LIN {X 0,Y 337.966,Z 536.674,A -85,B 0,C 180,E1 16019.152,E2 16019.152} C_VEL
LIN {X 0,Y 337.966,Z 536.674,A -85,B 0,C 180,E1 16014.908,E2 16014.908} C_VEL
LIN {X 0,Y 337.973,Z 536.675,A -85,B 0,C 180,E1 16010.807,E2 16010.807} C_VEL
LIN {X 0,Y 337.973,Z 536.677,A -85,B 0,C 180,E1 16006.484,E2 16006.484} C_VEL
LIN {X 0,Y 337.975,Z 536.732,A -85,B 0,C 180,E1 16002.259,E2 16002.259} C_VEL
LIN {X 0,Y 338.082,Z 537.452,A -85,B 0,C 180,E1 16001.73,E2 16001.73} C_VEL
LIN {X 0,Y 340.143,Z 542.274,A -85,B 0,C 180,E1 15999.651,E2 15999.651} C_VEL
LIN {X 0,Y 341.904,Z 546.345,A -85,B 0,C 180,E1 15998.017,E2 15998.017} C_VEL
LIN {X 0,Y 344.615,Z 552.699,A -85,B 0,C 180,E1 15995.632,E2 15995.632} C_VEL
LIN {X 0,Y 348.357,Z 562.803,A -85,B 0,C 180,E1 15992.291,E2 15992.291} C_VEL
LIN {X 0,Y 352.153,Z 574.379,A -85,B 0,C 180,E1 15988.885,E2 15988.885} C_VEL
LIN {X 0,Y 355.607,Z 586.974,A -85,B 0,C 180,E1 15985.587,E2 15985.587} C_VEL
LIN {X 0,Y 357.271,Z 594.978,A -85,B 0,C 180,E1 15983.697,E2 15983.697} C_VEL
LIN {X 0,Y 352.627,Z 621.546,A -85,B 0,C 180,E1 15979.08,E2 15979.08} C_VEL
LIN {X 0,Y 351.561,Z 628.87,A -85,B 0,C 180,E1 15977.84,E2 15977.84} C_VEL
LIN {X 0,Y 353.194,Z 637.289,A -85,B 0,C 180,E1 15977.353,E2 15977.353} C_VEL
LIN {X 0,Y 358.481,Z 665.393,A -85,B 0,C 180,E1 15976.019,E2 15976.019} C_VEL
LIN {X 0,Y 358.626,Z 670.018,A -85,B 0,C 180,E1 15975.886,E2 15975.886} C_VEL
LIN {X 0,Y 355.455,Z 759.785,A -85,B 0,C 180,E1 15973.88,E2 15973.88} C_VEL
LIN {X 0,Y 354.554,Z 775.918,A -85,B 0,C 180,E1 15973.222,E2 15973.222} C_VEL
LIN {X 0,Y 353.283,Z 790.634,A -85,B 0,C 180,E1 15972.337,E2 15972.337} C_VEL
LIN {X 0,Y 351.593,Z 804.794,A -85,B 0,C 180,E1 15971.173,E2 15971.173} C_VEL
LIN {X 0,Y 349.721,Z 817.611,A -85,B 0,C 180,E1 15969.816,E2 15969.816} C_VEL
LIN {X 0,Y 347.648,Z 829.608,A -85,B 0,C 180,E1 15968.19,E2 15968.19} C_VEL
LIN {X 0,Y 345.547,Z 840.726,A -85,B 0,C 180,E1 15966.286,E2 15966.286} C_VEL
LIN {X 0,Y 343.522,Z 850.351,A -85,B 0,C 180,E1 15964.171,E2 15964.171} C_VEL
LIN {X 0,Y 341.794,Z 858.2,A -85,B 0,C 180,E1 15961.965,E2 15961.965} C_VEL
LIN {X 0,Y 340.328,Z 864.589,A -85,B 0,C 180,E1 15959.57,E2 15959.57} C_VEL
LIN {X 0,Y 339.205,Z 869.505,A -85,B 0,C 180,E1 15956.992,E2 15956.992} C_VEL
LIN {X 0,Y 338.46,Z 872.53,A -85,B 0,C 180,E1 15954.425,E2 15954.425} C_VEL
LIN {X 0,Y 338.026,Z 873.979,A -85,B 0,C 180,E1 15951.695,E2 15951.695} C_VEL
LIN {X 0,Y 337.887,Z 873.587,A -85,B 0,C 180,E1 15948.992,E2 15948.992} C_VEL
LIN {X 0,Y 338.036,Z 871.502,A -85,B 0,C 180,E1 15946.316,E2 15946.316} C_VEL
LIN {X 0,Y 338.482,Z 867.484,A -85,B 0,C 180,E1 15943.625,E2 15943.625} C_VEL
LIN {X 0,Y 339.191,Z 862.191,A -85,B 0,C 180,E1 15941.216,E2 15941.216} C_VEL
LIN {X 0,Y 340.243,Z 854.856,A -85,B 0,C 180,E1 15938.787,E2 15938.787} C_VEL
LIN {X 0,Y 341.572,Z 846.059,A -85,B 0,C 180,E1 15936.553,E2 15936.553} C_VEL
LIN {X 0,Y 343.083,Z 835.74,A -85,B 0,C 180,E1 15934.511,E2 15934.511} C_VEL
LIN {X 0,Y 344.63,Z 824.489,A -85,B 0,C 180,E1 15932.742,E2 15932.742} C_VEL
LIN {X 0,Y 346.308,Z 810.951,A -85,B 0,C 180,E1 15931.073,E2 15931.073} C_VEL
LIN {X 0,Y 347.77,Z 796.978,A -85,B 0,C 180,E1 15929.751,E2 15929.751} C_VEL
LIN {X 0,Y 349.008,Z 782.059,A -85,B 0,C 180,E1 15928.685,E2 15928.685} C_VEL
LIN {X 0,Y 349.935,Z 765.507,A -85,B 0,C 180,E1 15927.869,E2 15927.869} C_VEL
LIN {X 0,Y 350.434,Z 748.757,A -85,B 0,C 180,E1 15927.374,E2 15927.374} C_VEL
LIN {X 0,Y 352.56,Z 663.643,A -85,B 0,C 180,E1 15925.551,E2 15925.551} C_VEL
LIN {X 0,Y 347.243,Z 631.526,A -85,B 0,C 180,E1 15924.385,E2 15924.385} C_VEL
LIN {X 0,Y 346.41,Z 628.646,A -85,B 0,C 180,E1 15924.113,E2 15924.113} C_VEL
LIN {X 0,Y 343.112,Z 619.723,A -85,B 0,C 180,E1 15922.259,E2 15922.259} C_VEL
LIN {X 0,Y 342.08,Z 612.242,A -85,B 0,C 180,E1 15920.819,E2 15920.819} C_VEL
LIN {X 0,Y 342.337,Z 607.788,A -85,B 0,C 180,E1 15920.058,E2 15920.058} C_VEL
LIN {X 0,Y 345.024,Z 588.546,A -85,B 0,C 180,E1 15916.765,E2 15916.765} C_VEL
LIN {X 0,Y 341.029,Z 572.719,A -85,B 0,C 180,E1 15913.301,E2 15913.301} C_VEL
LIN {X 0,Y 336.529,Z 557.319,A -85,B 0,C 180,E1 15909.658,E2 15909.658} C_VEL
LIN {X 0,Y 331.897,Z 543.403,A -85,B 0,C 180,E1 15906.097,E2 15906.097} C_VEL
LIN {X 0,Y 329.996,Z 537.777,A -85,B 0,C 180,E1 15904.469,E2 15904.469} C_VEL
LIN {X 0,Y 329.967,Z 537.621,A -85,B 0,C 180,E1 15900.07,E2 15900.07} C_VEL
LIN {X 0,Y 329.979,Z 537.693,A -85,B 0,C 180,E1 15895.696,E2 15895.696} C_VEL
LIN {X 0,Y 329.985,Z 537.683,A -85,B 0,C 180,E1 15891.379,E2 15891.379} C_VEL
LIN {X 0,Y 329.987,Z 537.665,A -85,B 0,C 180,E1 15887.161,E2 15887.161} C_VEL
LIN {X 0,Y 330.001,Z 537.675,A -85,B 0,C 180,E1 15882.845,E2 15882.845} C_VEL
LIN {X 0,Y 330.015,Z 537.684,A -85,B 0,C 180,E1 15878.589,E2 15878.589} C_VEL
LIN {X 0,Y 330.021,Z 537.65,A -85,B 0,C 180,E1 15874.201,E2 15874.201} C_VEL
LIN {X 0,Y 330.017,Z 537.688,A -85,B 0,C 180,E1 15869.794,E2 15869.794} C_VEL
LIN {X 0,Y 330.002,Z 537.65,A -85,B 0,C 180,E1 15865.464,E2 15865.464} C_VEL
LIN {X 0,Y 330.008,Z 537.687,A -85,B 0,C 180,E1 15861.32,E2 15861.32} C_VEL
LIN {X 0,Y 329.999,Z 537.646,A -85,B 0,C 180,E1 15857.092,E2 15857.092} C_VEL
LIN {X 0,Y 330.001,Z 537.689,A -85,B 0,C 180,E1 15852.779,E2 15852.779} C_VEL
LIN {X 0,Y 329.995,Z 537.643,A -85,B 0,C 180,E1 15848.363,E2 15848.363} C_VEL
LIN {X 0,Y 330.006,Z 537.688,A -85,B 0,C 180,E1 15843.996,E2 15843.996} C_VEL
LIN {X 0,Y 330.01,Z 537.645,A -85,B 0,C 180,E1 15839.653,E2 15839.653} C_VEL
LIN {X 0,Y 330.028,Z 537.683,A -85,B 0,C 180,E1 15835.308,E2 15835.308} C_VEL
LIN {X 0,Y 330.039,Z 537.658,A -85,B 0,C 180,E1 15830.958,E2 15830.958} C_VEL
LIN {X 0,Y 330.045,Z 537.667,A -85,B 0,C 180,E1 15826.689,E2 15826.689} C_VEL
LIN {X 0,Y 330.039,Z 537.688,A -85,B 0,C 180,E1 15822.365,E2 15822.365} C_VEL
LIN {X 0,Y 330.022,Z 537.666,A -85,B 0,C 180,E1 15817.977,E2 15817.977} C_VEL
LIN {X 0,Y 330.022,Z 537.665,A -85,B 0,C 180,E1 15813.733,E2 15813.733} C_VEL
LIN {X 0,Y 330.022,Z 537.675,A -85,B 0,C 180,E1 15809.605,E2 15809.605} C_VEL
LIN {X 0,Y 330.017,Z 537.676,A -85,B 0,C 180,E1 15805.279,E2 15805.279} C_VEL
LIN {X 0,Y 330.042,Z 537.839,A -85,B 0,C 180,E1 15800.842,E2 15800.842} C_VEL
LIN {X 0,Y 334.415,Z 549.082,A -85,B 0,C 180,E1 15798.184,E2 15798.184} C_VEL
LIN {X 0,Y 340.554,Z 565.504,A -85,B 0,C 180,E1 15794.724,E2 15794.724} C_VEL
LIN {X 0,Y 346.891,Z 584.231,A -85,B 0,C 180,E1 15791.211,E2 15791.211} C_VEL
LIN {X 0,Y 350.84,Z 596.806,A -85,B 0,C 180,E1 15789.036,E2 15789.036} C_VEL
LIN {X 0,Y 347.425,Z 618.655,A -85,B 0,C 180,E1 15786.45,E2 15786.45} C_VEL
LIN {X 0,Y 350.293,Z 650.391,A -85,B 0,C 180,E1 15785.474,E2 15785.474} C_VEL
LIN {X 0,Y 346.126,Z 809.723,A -85,B 0,C 180,E1 15782.248,E2 15782.248} C_VEL
LIN {X 0,Y 344.907,Z 828.121,A -85,B 0,C 180,E1 15781.593,E2 15781.593} C_VEL
LIN {X 0,Y 343.141,Z 845.982,A -85,B 0,C 180,E1 15780.658,E2 15780.658} C_VEL
LIN {X 0,Y 341.062,Z 863.504,A -85,B 0,C 180,E1 15779.409,E2 15779.409} C_VEL
LIN {X 0,Y 338.838,Z 880.035,A -85,B 0,C 180,E1 15777.885,E2 15777.885} C_VEL
LIN {X 0,Y 336.527,Z 895.631,A -85,B 0,C 180,E1 15776.086,E2 15776.086} C_VEL
LIN {X 0,Y 334.335,Z 910.232,A -85,B 0,C 180,E1 15773.999,E2 15773.999} C_VEL
LIN {X 0,Y 332.359,Z 923.739,A -85,B 0,C 180,E1 15771.63,E2 15771.63} C_VEL
LIN {X 0,Y 330.752,Z 935.755,A -85,B 0,C 180,E1 15769.056,E2 15769.056} C_VEL
LIN {X 0,Y 329.6,Z 946.565,A -85,B 0,C 180,E1 15766.206,E2 15766.206} C_VEL
LIN {X 0,Y 328.998,Z 955.237,A -85,B 0,C 180,E1 15763.355,E2 15763.355} C_VEL
LIN {X 0,Y 328.857,Z 962.428,A -85,B 0,C 180,E1 15760.335,E2 15760.335} C_VEL
LIN {X 0,Y 329.045,Z 967.721,A -85,B 0,C 180,E1 15757.334,E2 15757.334} C_VEL
LIN {X 0,Y 329.372,Z 971.066,A -85,B 0,C 180,E1 15754.529,E2 15754.529} C_VEL
LIN {X 0,Y 329.618,Z 972.901,A -85,B 0,C 180,E1 15751.74,E2 15751.74} C_VEL
LIN {X 0,Y 329.628,Z 973.257,A -85,B 0,C 180,E1 15748.959,E2 15748.959} C_VEL
LIN {X 0,Y 329.383,Z 972.149,A -85,B 0,C 180,E1 15746.173,E2 15746.173} C_VEL
LIN {X 0,Y 329,Z 969.367,A -85,B 0,C 180,E1 15743.196,E2 15743.196} C_VEL
LIN {X 0,Y 328.752,Z 964.926,A -85,B 0,C 180,E1 15740.197,E2 15740.197} C_VEL
LIN {X 0,Y 328.822,Z 958.744,A -85,B 0,C 180,E1 15737.178,E2 15737.178} C_VEL
LIN {X 0,Y 329.431,Z 950.694,A -85,B 0,C 180,E1 15734.151,E2 15734.151} C_VEL
LIN {X 0,Y 330.651,Z 940.705,A -85,B 0,C 180,E1 15731.17,E2 15731.17} C_VEL
LIN {X 0,Y 332.551,Z 928.756,A -85,B 0,C 180,E1 15728.3,E2 15728.3} C_VEL
LIN {X 0,Y 334.778,Z 916.276,A -85,B 0,C 180,E1 15725.852,E2 15725.852} C_VEL
LIN {X 0,Y 337.361,Z 902.358,A -85,B 0,C 180,E1 15723.609,E2 15723.609} C_VEL
LIN {X 0,Y 340.16,Z 887.505,A -85,B 0,C 180,E1 15721.665,E2 15721.665} C_VEL
LIN {X 0,Y 342.88,Z 871.764,A -85,B 0,C 180,E1 15720.005,E2 15720.005} C_VEL
LIN {X 0,Y 345.515,Z 854.96,A -85,B 0,C 180,E1 15718.614,E2 15718.614} C_VEL
LIN {X 0,Y 347.798,Z 837.868,A -85,B 0,C 180,E1 15717.534,E2 15717.534} C_VEL
LIN {X 0,Y 349.721,Z 819.606,A -85,B 0,C 180,E1 15716.712,E2 15716.712} C_VEL
LIN {X 0,Y 350.87,Z 800.729,A -85,B 0,C 180,E1 15716.159,E2 15716.159} C_VEL
LIN {X 0,Y 355.558,Z 648.305,A -85,B 0,C 180,E1 15713.007,E2 15713.007} C_VEL
LIN {X 0,Y 352.568,Z 619.487,A -85,B 0,C 180,E1 15711.903,E2 15711.903} C_VEL
LIN {X 0,Y 355.795,Z 602.812,A -85,B 0,C 180,E1 15709.851,E2 15709.851} C_VEL
LIN {X 0,Y 351.503,Z 588.783,A -85,B 0,C 180,E1 15706.953,E2 15706.953} C_VEL
LIN {X 0,Y 346.879,Z 575.902,A -85,B 0,C 180,E1 15703.903,E2 15703.903} C_VEL
LIN {X 0,Y 342.361,Z 564.804,A -85,B 0,C 180,E1 15700.858,E2 15700.858} C_VEL
LIN {X 0,Y 338.122,Z 554.907,A -85,B 0,C 180,E1 15697.743,E2 15697.743} C_VEL
LIN {X 0,Y 334.128,Z 546.479,A -85,B 0,C 180,E1 15694.632,E2 15694.632} C_VEL
LIN {X 0,Y 331.778,Z 541.799,A -85,B 0,C 180,E1 15692.645,E2 15692.645} C_VEL
LIN {X 0,Y 330.017,Z 537.816,A -85,B 0,C 180,E1 15690.743,E2 15690.743} C_VEL
LIN {X 0,Y 330,Z 537.683,A -85,B 0,C 180,E1 15686.448,E2 15686.448} C_VEL
LIN {X 0,Y 329.997,Z 537.68,A -85,B 0,C 180,E1 15682.255,E2 15682.255} C_VEL
LIN {X 0,Y 330.002,Z 537.674,A -85,B 0,C 180,E1 15677.963,E2 15677.963} C_VEL
LIN {X 0,Y 330.008,Z 537.665,A -85,B 0,C 180,E1 15673.669,E2 15673.669} C_VEL
LIN {X 0,Y 330.009,Z 537.663,A -85,B 0,C 180,E1 15669.24,E2 15669.24} C_VEL
LIN {X 0,Y 330.01,Z 537.663,A -85,B 0,C 180,E1 15665.04,E2 15665.04} C_VEL
LIN {X 0,Y 330.004,Z 537.668,A -85,B 0,C 180,E1 15660.694,E2 15660.694} C_VEL
LIN {X 0,Y 330.005,Z 537.679,A -85,B 0,C 180,E1 15656.526,E2 15656.526} C_VEL
LIN {X 0,Y 330.003,Z 537.683,A -85,B 0,C 180,E1 15652.153,E2 15652.153} C_VEL
LIN {X 0,Y 330.003,Z 537.681,A -85,B 0,C 180,E1 15647.755,E2 15647.755} C_VEL
LIN {X 0,Y 330.064,Z 537.971,A -85,B 0,C 180,E1 15644.212,E2 15644.212} C_VEL
LIN {X 0,Y 331.804,Z 541.827,A -85,B 0,C 180,E1 15642.28,E2 15642.28} C_VEL
LIN {X 0,Y 334.221,Z 547.755,A -85,B 0,C 180,E1 15639.694,E2 15639.694} C_VEL
LIN {X 0,Y 335.816,Z 551.504,A -85,B 0,C 180,E1 15638.15,E2 15638.15} C_VEL
LIN {X 0,Y 338.592,Z 558.281,A -85,B 0,C 180,E1 15635.58,E2 15635.58} C_VEL
LIN {X 0,Y 341.924,Z 567.424,A -85,B 0,C 180,E1 15632.482,E2 15632.482} C_VEL
LIN {X 0,Y 345.652,Z 579.019,A -85,B 0,C 180,E1 15629.009,E2 15629.009} C_VEL
LIN {X 0,Y 349.02,Z 591.691,A -85,B 0,C 180,E1 15625.642,E2 15625.642} C_VEL
LIN {X 0,Y 350.297,Z 597.841,A -85,B 0,C 180,E1 15624.147,E2 15624.147} C_VEL
LIN {X 0,Y 345.407,Z 624.426,A -85,B 0,C 180,E1 15619.443,E2 15619.443} C_VEL
LIN {X 0,Y 344.818,Z 629.173,A -85,B 0,C 180,E1 15618.67,E2 15618.67} C_VEL
LIN {X 0,Y 350.44,Z 657.682,A -85,B 0,C 180,E1 15617.166,E2 15617.166} C_VEL
LIN {X 0,Y 352.161,Z 669.248,A -85,B 0,C 180,E1 15616.658,E2 15616.658} C_VEL
LIN {X 0,Y 348.762,Z 760.258,A -85,B 0,C 180,E1 15614.589,E2 15614.589} C_VEL
LIN {X 0,Y 347.832,Z 776.174,A -85,B 0,C 180,E1 15613.935,E2 15613.935} C_VEL
LIN {X 0,Y 346.483,Z 791.091,A -85,B 0,C 180,E1 15613.03,E2 15613.03} C_VEL
LIN {X 0,Y 344.607,Z 806.014,A -85,B 0,C 180,E1 15611.782,E2 15611.782} C_VEL
LIN {X 0,Y 342.6,Z 818.978,A -85,B 0,C 180,E1 15610.376,E2 15610.376} C_VEL
LIN {X 0,Y 340.257,Z 831.741,A -85,B 0,C 180,E1 15608.587,E2 15608.587} C_VEL
LIN {X 0,Y 338.087,Z 842.463,A -85,B 0,C 180,E1 15606.677,E2 15606.677} C_VEL
LIN {X 0,Y 335.889,Z 852.281,A -85,B 0,C 180,E1 15604.437,E2 15604.437} C_VEL
LIN {X 0,Y 334.013,Z 860.185,A -85,B 0,C 180,E1 15602.096,E2 15602.096} C_VEL
LIN {X 0,Y 332.444,Z 866.583,A -85,B 0,C 180,E1 15599.549,E2 15599.549} C_VEL
LIN {X 0,Y 331.287,Z 871.197,A -85,B 0,C 180,E1 15596.913,E2 15596.913} C_VEL
LIN {X 0,Y 330.495,Z 874.156,A -85,B 0,C 180,E1 15594.101,E2 15594.101} C_VEL
LIN {X 0,Y 330.077,Z 875.213,A -85,B 0,C 180,E1 15591.311,E2 15591.311} C_VEL
LIN {X 0,Y 329.981,Z 874.51,A -85,B 0,C 180,E1 15588.484,E2 15588.484} C_VEL
LIN {X 0,Y 330.197,Z 871.886,A -85,B 0,C 180,E1 15585.649,E2 15585.649} C_VEL
LIN {X 0,Y 330.693,Z 867.877,A -85,B 0,C 180,E1 15583.103,E2 15583.103} C_VEL
LIN {X 0,Y 331.566,Z 861.643,A -85,B 0,C 180,E1 15580.421,E2 15580.421} C_VEL
LIN {X 0,Y 332.679,Z 854.467,A -85,B 0,C 180,E1 15578.118,E2 15578.118} C_VEL
LIN {X 0,Y 334.125,Z 845.202,A -85,B 0,C 180,E1 15575.837,E2 15575.837} C_VEL
LIN {X 0,Y 335.704,Z 834.859,A -85,B 0,C 180,E1 15573.827,E2 15573.827} C_VEL
LIN {X 0,Y 337.509,Z 821.953,A -85,B 0,C 180,E1 15571.865,E2 15571.865} C_VEL
LIN {X 0,Y 339.128,Z 809,A -85,B 0,C 180,E1 15570.336,E2 15570.336} C_VEL
LIN {X 0,Y 340.673,Z 794.254,A -85,B 0,C 180,E1 15568.989,E2 15568.989} C_VEL
LIN {X 0,Y 341.907,Z 778.574,A -85,B 0,C 180,E1 15567.945,E2 15567.945} C_VEL
LIN {X 0,Y 342.723,Z 762.988,A -85,B 0,C 180,E1 15567.234,E2 15567.234} C_VEL
LIN {X 0,Y 343.35,Z 740.557,A -85,B 0,C 180,E1 15566.649,E2 15566.649} C_VEL
LIN {X 0,Y 345.34,Z 664.762,A -85,B 0,C 180,E1 15565,E2 15565} C_VEL
LIN {X 0,Y 339.575,Z 629.437,A -85,B 0,C 180,E1 15563.659,E2 15563.659} C_VEL
LIN {X 0,Y 340.187,Z 623.578,A -85,B 0,C 180,E1 15562.738,E2 15562.738} C_VEL
LIN {X 0,Y 342.337,Z 607.788,A -85,B 0,C 180,E1 15560.058,E2 15560.058} C_VEL
LIN {X 0,Y 342.242,Z 602.599,A -85,B 0,C 180,E1 15559.093,E2 15559.093} C_VEL
LIN {X 0,Y 340.148,Z 595.894,A -85,B 0,C 180,E1 15557.63,E2 15557.63} C_VEL
LIN {X 0,Y 336.388,Z 586.056,A -85,B 0,C 180,E1 15555.351,E2 15555.351} C_VEL
LIN {X 0,Y 332.439,Z 570.926,A -85,B 0,C 180,E1 15551.883,E2 15551.883} C_VEL
LIN {X 0,Y 328.118,Z 556.573,A -85,B 0,C 180,E1 15548.345,E2 15548.345} C_VEL
LIN {X 0,Y 323.866,Z 544.068,A -85,B 0,C 180,E1 15544.979,E2 15544.979} C_VEL
LIN {X 0,Y 322.078,Z 538.78,A -85,B 0,C 180,E1 15543.39,E2 15543.39} C_VEL
LIN {X 0,Y 322.071,Z 538.601,A -85,B 0,C 180,E1 15538.98,E2 15538.98} C_VEL
LIN {X 0,Y 322.06,Z 538.676,A -85,B 0,C 180,E1 15534.511,E2 15534.511} C_VEL
LIN {X 0,Y 322.056,Z 538.683,A -85,B 0,C 180,E1 15530.243,E2 15530.243} C_VEL
LIN {X 0,Y 322.05,Z 538.664,A -85,B 0,C 180,E1 15525.939,E2 15525.939} C_VEL
LIN {X 0,Y 322.042,Z 538.649,A -85,B 0,C 180,E1 15521.564,E2 15521.564} C_VEL
LIN {X 0,Y 322.051,Z 538.681,A -85,B 0,C 180,E1 15517.073,E2 15517.073} C_VEL
LIN {X 0,Y 322.059,Z 538.651,A -85,B 0,C 180,E1 15512.698,E2 15512.698} C_VEL
LIN {X 0,Y 322.065,Z 538.665,A -85,B 0,C 180,E1 15508.533,E2 15508.533} C_VEL
LIN {X 0,Y 322.081,Z 538.655,A -85,B 0,C 180,E1 15504.127,E2 15504.127} C_VEL
LIN {X 0,Y 322.09,Z 538.657,A -85,B 0,C 180,E1 15499.855,E2 15499.855} C_VEL
LIN {X 0,Y 322.091,Z 538.651,A -85,B 0,C 180,E1 15495.484,E2 15495.484} C_VEL
LIN {X 0,Y 322.075,Z 538.659,A -85,B 0,C 180,E1 15491.098,E2 15491.098} C_VEL
LIN {X 0,Y 322.066,Z 538.651,A -85,B 0,C 180,E1 15486.775,E2 15486.775} C_VEL
LIN {X 0,Y 322.064,Z 538.658,A -85,B 0,C 180,E1 15482.491,E2 15482.491} C_VEL
LIN {X 0,Y 322.064,Z 538.663,A -85,B 0,C 180,E1 15478.043,E2 15478.043} C_VEL
LIN {X 0,Y 322.066,Z 538.65,A -85,B 0,C 180,E1 15473.762,E2 15473.762} C_VEL
LIN {X 0,Y 322.077,Z 538.674,A -85,B 0,C 180,E1 15469.446,E2 15469.446} C_VEL
LIN {X 0,Y 322.089,Z 538.643,A -85,B 0,C 180,E1 15465.069,E2 15465.069} C_VEL
LIN {X 0,Y 322.104,Z 538.665,A -85,B 0,C 180,E1 15460.668,E2 15460.668} C_VEL
LIN {X 0,Y 322.107,Z 538.676,A -85,B 0,C 180,E1 15456.301,E2 15456.301} C_VEL
LIN {X 0,Y 322.093,Z 538.666,A -85,B 0,C 180,E1 15451.832,E2 15451.832} C_VEL
LIN {X 0,Y 322.086,Z 538.665,A -85,B 0,C 180,E1 15447.517,E2 15447.517} C_VEL
LIN {X 0,Y 322.083,Z 538.671,A -85,B 0,C 180,E1 15443.192,E2 15443.192} C_VEL
LIN {X 0,Y 322.168,Z 539.03,A -85,B 0,C 180,E1 15441.887,E2 15441.887} C_VEL
LIN {X 0,Y 327.939,Z 553.754,A -85,B 0,C 180,E1 15438.344,E2 15438.344} C_VEL
LIN {X 0,Y 333.871,Z 569.79,A -85,B 0,C 180,E1 15434.907,E2 15434.907} C_VEL
LIN {X 0,Y 340.129,Z 588.566,A -85,B 0,C 180,E1 15431.316,E2 15431.316} C_VEL
LIN {X 0,Y 343.403,Z 599.528,A -85,B 0,C 180,E1 15429.399,E2 15429.399} C_VEL
LIN {X 0,Y 340.255,Z 618.442,A -85,B 0,C 180,E1 15427.094,E2 15427.094} C_VEL
LIN {X 0,Y 343.117,Z 651.293,A -85,B 0,C 180,E1 15426.05,E2 15426.05} C_VEL
LIN {X 0,Y 338.797,Z 809.111,A -85,B 0,C 180,E1 15422.792,E2 15422.792} C_VEL
LIN {X 0,Y 337.541,Z 827.487,A -85,B 0,C 180,E1 15422.124,E2 15422.124} C_VEL
LIN {X 0,Y 335.706,Z 845.479,A -85,B 0,C 180,E1 15421.164,E2 15421.164} C_VEL
LIN {X 0,Y 333.622,Z 862.449,A -85,B 0,C 180,E1 15419.933,E2 15419.933} C_VEL
LIN {X 0,Y 331.31,Z 879.057,A -85,B 0,C 180,E1 15418.38,E2 15418.38} C_VEL
LIN {X 0,Y 328.911,Z 894.705,A -85,B 0,C 180,E1 15416.543,E2 15416.543} C_VEL
LIN {X 0,Y 326.614,Z 909.308,A -85,B 0,C 180,E1 15414.411,E2 15414.411} C_VEL
LIN {X 0,Y 324.553,Z 922.821,A -85,B 0,C 180,E1 15411.983,E2 15411.983} C_VEL
LIN {X 0,Y 322.873,Z 934.797,A -85,B 0,C 180,E1 15409.351,E2 15409.351} C_VEL
LIN {X 0,Y 321.67,Z 945.585,A -85,B 0,C 180,E1 15406.432,E2 15406.432} C_VEL
LIN {X 0,Y 321.038,Z 954.233,A -85,B 0,C 180,E1 15403.509,E2 15403.509} C_VEL
LIN {X 0,Y 320.897,Z 961.397,A -85,B 0,C 180,E1 15400.413,E2 15400.413} C_VEL
LIN {X 0,Y 321.105,Z 966.658,A -85,B 0,C 180,E1 15397.336,E2 15397.336} C_VEL
LIN {X 0,Y 321.474,Z 970.135,A -85,B 0,C 180,E1 15394.283,E2 15394.283} C_VEL
LIN {X 0,Y 321.721,Z 971.821,A -85,B 0,C 180,E1 15391.427,E2 15391.427} C_VEL
LIN {X 0,Y 321.693,Z 972.013,A -85,B 0,C 180,E1 15388.577,E2 15388.577} C_VEL
LIN {X 0,Y 321.372,Z 970.6,A -85,B 0,C 180,E1 15385.542,E2 15385.542} C_VEL
LIN {X 0,Y 320.964,Z 967.538,A -85,B 0,C 180,E1 15382.485,E2 15382.485} C_VEL
LIN {X 0,Y 320.755,Z 962.473,A -85,B 0,C 180,E1 15379.224,E2 15379.224} C_VEL
LIN {X 0,Y 321.002,Z 955.444,A -85,B 0,C 180,E1 15375.943,E2 15375.943} C_VEL
LIN {X 0,Y 321.865,Z 946.847,A -85,B 0,C 180,E1 15372.839,E2 15372.839} C_VEL
LIN {X 0,Y 323.333,Z 936.79,A -85,B 0,C 180,E1 15369.929,E2 15369.929} C_VEL
LIN {X 0,Y 325.414,Z 925.119,A -85,B 0,C 180,E1 15367.186,E2 15367.186} C_VEL
LIN {X 0,Y 327.971,Z 911.791,A -85,B 0,C 180,E1 15364.643,E2 15364.643} C_VEL
LIN {X 0,Y 330.77,Z 897.738,A -85,B 0,C 180,E1 15362.457,E2 15362.457} C_VEL
LIN {X 0,Y 333.812,Z 882.055,A -85,B 0,C 180,E1 15360.486,E2 15360.486} C_VEL
LIN {X 0,Y 336.643,Z 866.134,A -85,B 0,C 180,E1 15358.888,E2 15358.888} C_VEL
LIN {X 0,Y 339.3,Z 849.353,A -85,B 0,C 180,E1 15357.572,E2 15357.572} C_VEL
LIN {X 0,Y 341.59,Z 832.287,A -85,B 0,C 180,E1 15356.569,E2 15356.569} C_VEL
LIN {X 0,Y 343.399,Z 813.982,A -85,B 0,C 180,E1 15355.808,E2 15355.808} C_VEL
LIN {X 0,Y 344.383,Z 794.102,A -85,B 0,C 180,E1 15355.297,E2 15355.297} C_VEL
LIN {X 0,Y 349.099,Z 649.224,A -85,B 0,C 180,E1 15352.248,E2 15352.248} C_VEL
LIN {X 0,Y 346.068,Z 619.537,A -85,B 0,C 180,E1 15351.07,E2 15351.07} C_VEL
LIN {X 0,Y 348.804,Z 605.663,A -85,B 0,C 180,E1 15349.318,E2 15349.318} C_VEL
LIN {X 0,Y 344.569,Z 591.717,A -85,B 0,C 180,E1 15346.328,E2 15346.328} C_VEL
LIN {X 0,Y 339.815,Z 578.458,A -85,B 0,C 180,E1 15343.049,E2 15343.049} C_VEL
LIN {X 0,Y 335.347,Z 567.434,A -85,B 0,C 180,E1 15339.869,E2 15339.869} C_VEL
LIN {X 0,Y 331.458,Z 558.711,A -85,B 0,C 180,E1 15336.939,E2 15336.939} C_VEL
LIN {X 0,Y 328.271,Z 551.753,A -85,B 0,C 180,E1 15334.296,E2 15334.296} C_VEL
LIN {X 0,Y 326.185,Z 547.428,A -85,B 0,C 180,E1 15332.441,E2 15332.441} C_VEL
LIN {X 0,Y 323.808,Z 542.721,A -85,B 0,C 180,E1 15330.177,E2 15330.177} C_VEL
LIN {X 0,Y 322.118,Z 538.913,A -85,B 0,C 180,E1 15328.152,E2 15328.152} C_VEL
LIN {X 0,Y 322.087,Z 538.652,A -85,B 0,C 180,E1 15323.701,E2 15323.701} C_VEL
LIN {X 0,Y 322.074,Z 538.652,A -85,B 0,C 180,E1 15319.401,E2 15319.401} C_VEL
LIN {X 0,Y 322.059,Z 538.654,A -85,B 0,C 180,E1 15315.115,E2 15315.115} C_VEL
LIN {X 0,Y 322.043,Z 538.662,A -85,B 0,C 180,E1 15310.736,E2 15310.736} C_VEL
LIN {X 0,Y 322.041,Z 538.674,A -85,B 0,C 180,E1 15306.417,E2 15306.417} C_VEL
LIN {X 0,Y 322.049,Z 538.682,A -85,B 0,C 180,E1 15301.957,E2 15301.957} C_VEL
LIN {X 0,Y 322.058,Z 538.678,A -85,B 0,C 180,E1 15297.687,E2 15297.687} C_VEL
LIN {X 0,Y 322.073,Z 538.669,A -85,B 0,C 180,E1 15293.364,E2 15293.364} C_VEL
LIN {X 0,Y 322.083,Z 538.665,A -85,B 0,C 180,E1 15289.084,E2 15289.084} C_VEL
LIN {X 0,Y 322.147,Z 538.996,A -85,B 0,C 180,E1 15286.859,E2 15286.859} C_VEL
LIN {X 0,Y 323.769,Z 542.656,A -85,B 0,C 180,E1 15284.781,E2 15284.781} C_VEL
LIN {X 0,Y 326.234,Z 548.245,A -85,B 0,C 180,E1 15281.967,E2 15281.967} C_VEL
LIN {X 0,Y 328.203,Z 552.937,A -85,B 0,C 180,E1 15279.864,E2 15279.864} C_VEL
LIN {X 0,Y 330.748,Z 558.738,A -85,B 0,C 180,E1 15277.423,E2 15277.423} C_VEL
LIN {X 0,Y 334.632,Z 569.451,A -85,B 0,C 180,E1 15273.563,E2 15273.563} C_VEL
LIN {X 0,Y 338.085,Z 579.995,A -85,B 0,C 180,E1 15270.208,E2 15270.208} C_VEL
LIN {X 0,Y 341.315,Z 591.804,A -85,B 0,C 180,E1 15266.899,E2 15266.899} C_VEL
LIN {X 0,Y 343.312,Z 600.922,A -85,B 0,C 180,E1 15264.58,E2 15264.58} C_VEL
LIN {X 0,Y 338.273,Z 627.02,A -85,B 0,C 180,E1 15259.882,E2 15259.882} C_VEL
LIN {X 0,Y 338.081,Z 628.557,A -85,B 0,C 180,E1 15259.632,E2 15259.632} C_VEL
LIN {X 0,Y 340.225,Z 639.451,A -85,B 0,C 180,E1 15258.969,E2 15258.969} C_VEL
LIN {X 0,Y 345.236,Z 666.408,A -85,B 0,C 180,E1 15257.586,E2 15257.586} C_VEL
LIN {X 0,Y 345.671,Z 671.031,A -85,B 0,C 180,E1 15257.406,E2 15257.406} C_VEL
LIN {X 0,Y 342.148,Z 760.993,A -85,B 0,C 180,E1 15255.326,E2 15255.326} C_VEL
LIN {X 0,Y 341.156,Z 777.024,A -85,B 0,C 180,E1 15254.654,E2 15254.654} C_VEL
LIN {X 0,Y 339.676,Z 792.431,A -85,B 0,C 180,E1 15253.698,E2 15253.698} C_VEL
LIN {X 0,Y 337.727,Z 807.04,A -85,B 0,C 180,E1 15252.447,E2 15252.447} C_VEL
LIN {X 0,Y 335.523,Z 820.41,A -85,B 0,C 180,E1 15250.958,E2 15250.958} C_VEL
LIN {X 0,Y 332.992,Z 833.393,A -85,B 0,C 180,E1 15249.084,E2 15249.084} C_VEL
LIN {X 0,Y 330.762,Z 843.69,A -85,B 0,C 180,E1 15247.192,E2 15247.192} C_VEL
LIN {X 0,Y 328.435,Z 853.473,A -85,B 0,C 180,E1 15244.907,E2 15244.907} C_VEL
LIN {X 0,Y 326.509,Z 861.103,A -85,B 0,C 180,E1 15242.607,E2 15242.607} C_VEL
LIN {X 0,Y 324.758,Z 867.748,A -85,B 0,C 180,E1 15239.913,E2 15239.913} C_VEL
LIN {X 0,Y 323.512,Z 872.366,A -85,B 0,C 180,E1 15237.215,E2 15237.215} C_VEL
LIN {X 0,Y 322.645,Z 875.33,A -85,B 0,C 180,E1 15234.336,E2 15234.336} C_VEL
LIN {X 0,Y 322.182,Z 876.407,A -85,B 0,C 180,E1 15231.477,E2 15231.477} C_VEL
LIN {X 0,Y 322.059,Z 875.75,A -85,B 0,C 180,E1 15228.645,E2 15228.645} C_VEL
LIN {X 0,Y 322.251,Z 873.335,A -85,B 0,C 180,E1 15225.842,E2 15225.842} C_VEL
LIN {X 0,Y 322.78,Z 869.153,A -85,B 0,C 180,E1 15223.066,E2 15223.066} C_VEL
LIN {X 0,Y 323.61,Z 863.456,A -85,B 0,C 180,E1 15220.5,E2 15220.5} C_VEL
LIN {X 0,Y 324.832,Z 855.866,A -85,B 0,C 180,E1 15217.959,E2 15217.959} C_VEL
LIN {X 0,Y 326.329,Z 846.691,A -85,B 0,C 180,E1 15215.624,E2 15215.624} C_VEL
LIN {X 0,Y 328.03,Z 836.05,A -85,B 0,C 180,E1 15213.493,E2 15213.493} C_VEL
LIN {X 0,Y 329.831,Z 823.712,A -85,B 0,C 180,E1 15211.561,E2 15211.561} C_VEL
LIN {X 0,Y 331.51,Z 811.033,A -85,B 0,C 180,E1 15209.998,E2 15209.998} C_VEL
LIN {X 0,Y 333.107,Z 796.594,A -85,B 0,C 180,E1 15208.622,E2 15208.622} C_VEL
LIN {X 0,Y 334.394,Z 781.562,A -85,B 0,C 180,E1 15207.556,E2 15207.556} C_VEL
LIN {X 0,Y 335.357,Z 765.231,A -85,B 0,C 180,E1 15206.751,E2 15206.751} C_VEL
LIN {X 0,Y 335.948,Z 745.23,A -85,B 0,C 180,E1 15206.188,E2 15206.188} C_VEL
LIN {X 0,Y 338.132,Z 665.713,A -85,B 0,C 180,E1 15204.42,E2 15204.42} C_VEL
LIN {X 0,Y 332.227,Z 629.211,A -85,B 0,C 180,E1 15202.998,E2 15202.998} C_VEL
LIN {X 0,Y 335.745,Z 603.789,A -85,B 0,C 180,E1 15198.664,E2 15198.664} C_VEL
LIN {X 0,Y 337.628,Z 591.171,A -85,B 0,C 180,E1 15196.469,E2 15196.469} C_VEL
LIN {X 0,Y 336.388,Z 586.056,A -85,B 0,C 180,E1 15195.351,E2 15195.351} C_VEL
LIN {X 0,Y 334.734,Z 582.402,A -85,B 0,C 180,E1 15194.446,E2 15194.446} C_VEL
LIN {X 0,Y 330.136,Z 577.467,A -85,B 0,C 180,E1 15192.909,E2 15192.909} C_VEL
LIN {X 0,Y 325.143,Z 572.083,A -85,B 0,C 180,E1 15191.165,E2 15191.165} C_VEL
LIN {X 0,Y 323.813,Z 569.083,A -85,B 0,C 180,E1 15190.363,E2 15190.363} C_VEL
LIN {X 0,Y 319.295,Z 554.495,A -85,B 0,C 180,E1 15186.566,E2 15186.566} C_VEL
LIN {X 0,Y 314.845,Z 542.103,A -85,B 0,C 180,E1 15182.991,E2 15182.991} C_VEL
LIN {X 0,Y 314.12,Z 539.792,A -85,B 0,C 180,E1 15182.239,E2 15182.239} C_VEL
LIN {X 0,Y 314.09,Z 539.606,A -85,B 0,C 180,E1 15177.863,E2 15177.863} C_VEL
LIN {X 0,Y 314.104,Z 539.651,A -85,B 0,C 180,E1 15173.47,E2 15173.47} C_VEL
LIN {X 0,Y 314.11,Z 539.662,A -85,B 0,C 180,E1 15169.253,E2 15169.253} C_VEL
LIN {X 0,Y 314.131,Z 539.667,A -85,B 0,C 180,E1 15164.784,E2 15164.784} C_VEL
LIN {X 0,Y 314.14,Z 539.635,A -85,B 0,C 180,E1 15160.25,E2 15160.25} C_VEL
LIN {X 0,Y 314.126,Z 539.648,A -85,B 0,C 180,E1 15155.851,E2 15155.851} C_VEL
LIN {X 0,Y 314.119,Z 539.66,A -85,B 0,C 180,E1 15151.458,E2 15151.458} C_VEL
LIN {X 0,Y 314.111,Z 539.629,A -85,B 0,C 180,E1 15146.971,E2 15146.971} C_VEL
LIN {X 0,Y 314.124,Z 539.666,A -85,B 0,C 180,E1 15142.456,E2 15142.456} C_VEL
LIN {X 0,Y 314.138,Z 539.618,A -85,B 0,C 180,E1 15137.984,E2 15137.984} C_VEL
LIN {X 0,Y 314.16,Z 539.664,A -85,B 0,C 180,E1 15133.622,E2 15133.622} C_VEL
LIN {X 0,Y 314.14,Z 539.615,A -85,B 0,C 180,E1 15129.158,E2 15129.158} C_VEL
LIN {X 0,Y 314.141,Z 539.665,A -85,B 0,C 180,E1 15124.93,E2 15124.93} C_VEL
LIN {X 0,Y 314.127,Z 539.618,A -85,B 0,C 180,E1 15120.547,E2 15120.547} C_VEL
LIN {X 0,Y 314.129,Z 539.668,A -85,B 0,C 180,E1 15116.168,E2 15116.168} C_VEL
LIN {X 0,Y 314.126,Z 539.628,A -85,B 0,C 180,E1 15111.765,E2 15111.765} C_VEL
LIN {X 0,Y 314.141,Z 539.655,A -85,B 0,C 180,E1 15107.314,E2 15107.314} C_VEL
LIN {X 0,Y 314.154,Z 539.657,A -85,B 0,C 180,E1 15102.974,E2 15102.974} C_VEL
LIN {X 0,Y 314.172,Z 539.634,A -85,B 0,C 180,E1 15098.532,E2 15098.532} C_VEL
LIN {X 0,Y 314.163,Z 539.641,A -85,B 0,C 180,E1 15094.15,E2 15094.15} C_VEL
LIN {X 0,Y 314.155,Z 539.653,A -85,B 0,C 180,E1 15089.811,E2 15089.811} C_VEL
LIN {X 0,Y 314.145,Z 539.654,A -85,B 0,C 180,E1 15085.491,E2 15085.491} C_VEL
LIN {X 0,Y 314.178,Z 539.907,A -85,B 0,C 180,E1 15083.144,E2 15083.144} C_VEL
LIN {X 0,Y 319.631,Z 553.552,A -85,B 0,C 180,E1 15079.645,E2 15079.645} C_VEL
LIN {X 0,Y 325.59,Z 569.497,A -85,B 0,C 180,E1 15076.051,E2 15076.051} C_VEL
LIN {X 0,Y 331.552,Z 587.178,A -85,B 0,C 180,E1 15072.492,E2 15072.492} C_VEL
LIN {X 0,Y 336.023,Z 601.859,A -85,B 0,C 180,E1 15069.821,E2 15069.821} C_VEL
LIN {X 0,Y 333.119,Z 618.895,A -85,B 0,C 180,E1 15067.72,E2 15067.72} C_VEL
LIN {X 0,Y 335.981,Z 652.102,A -85,B 0,C 180,E1 15066.651,E2 15066.651} C_VEL
LIN {X 0,Y 331.502,Z 808.449,A -85,B 0,C 180,E1 15063.361,E2 15063.361} C_VEL
LIN {X 0,Y 330.202,Z 826.887,A -85,B 0,C 180,E1 15062.678,E2 15062.678} C_VEL
LIN {X 0,Y 328.298,Z 844.95,A -85,B 0,C 180,E1 15061.692,E2 15061.692} C_VEL
LIN {X 0,Y 326.069,Z 862.383,A -85,B 0,C 180,E1 15060.394,E2 15060.394} C_VEL
LIN {X 0,Y 323.683,Z 878.838,A -85,B 0,C 180,E1 15058.808,E2 15058.808} C_VEL
LIN {X 0,Y 321.206,Z 894.345,A -85,B 0,C 180,E1 15056.931,E2 15056.931} C_VEL
LIN {X 0,Y 318.824,Z 908.839,A -85,B 0,C 180,E1 15054.751,E2 15054.751} C_VEL
LIN {X 0,Y 316.691,Z 922.298,A -85,B 0,C 180,E1 15052.264,E2 15052.264} C_VEL
LIN {X 0,Y 314.88,Z 934.783,A -85,B 0,C 180,E1 15049.424,E2 15049.424} C_VEL
LIN {X 0,Y 313.683,Z 945.217,A -85,B 0,C 180,E1 15046.481,E2 15046.481} C_VEL
LIN {X 0,Y 313.056,Z 953.719,A -85,B 0,C 180,E1 15043.484,E2 15043.484} C_VEL
LIN {X 0,Y 312.942,Z 960.865,A -85,B 0,C 180,E1 15040.242,E2 15040.242} C_VEL
LIN {X 0,Y 313.184,Z 965.855,A -85,B 0,C 180,E1 15037.154,E2 15037.154} C_VEL
LIN {X 0,Y 313.583,Z 969.192,A -85,B 0,C 180,E1 15034.024,E2 15034.024} C_VEL
LIN {X 0,Y 313.82,Z 970.734,A -85,B 0,C 180,E1 15031.097,E2 15031.097} C_VEL
LIN {X 0,Y 313.746,Z 970.763,A -85,B 0,C 180,E1 15028.176,E2 15028.176} C_VEL
LIN {X 0,Y 313.396,Z 969.311,A -85,B 0,C 180,E1 15025.244,E2 15025.244} C_VEL
LIN {X 0,Y 312.958,Z 966.104,A -85,B 0,C 180,E1 15022.056,E2 15022.056} C_VEL
LIN {X 0,Y 312.773,Z 961.014,A -85,B 0,C 180,E1 15018.758,E2 15018.758} C_VEL
LIN {X 0,Y 313.113,Z 953.847,A -85,B 0,C 180,E1 15015.367,E2 15015.367} C_VEL
LIN {X 0,Y 314.14,Z 944.953,A -85,B 0,C 180,E1 15012.113,E2 15012.113} C_VEL
LIN {X 0,Y 315.884,Z 934.277,A -85,B 0,C 180,E1 15009.028,E2 15009.028} C_VEL
LIN {X 0,Y 318.152,Z 922.554,A -85,B 0,C 180,E1 15006.285,E2 15006.285} C_VEL
LIN {X 0,Y 320.891,Z 909.235,A -85,B 0,C 180,E1 15003.744,E2 15003.744} C_VEL
LIN {X 0,Y 323.927,Z 894.89,A -85,B 0,C 180,E1 15001.523,E2 15001.523} C_VEL
LIN {X 0,Y 327.036,Z 879.596,A -85,B 0,C 180,E1 14999.608,E2 14999.608} C_VEL
LIN {X 0,Y 330.049,Z 863.397,A -85,B 0,C 180,E1 14997.99,E2 14997.99} C_VEL
LIN {X 0,Y 332.88,Z 846.127,A -85,B 0,C 180,E1 14996.661,E2 14996.661} C_VEL
LIN {X 0,Y 335.245,Z 828.475,A -85,B 0,C 180,E1 14995.662,E2 14995.662} C_VEL
LIN {X 0,Y 336.974,Z 810.197,A -85,B 0,C 180,E1 14994.948,E2 14994.948} C_VEL
LIN {X 0,Y 338.061,Z 784.928,A -85,B 0,C 180,E1 14994.349,E2 14994.349} C_VEL
LIN {X 0,Y 342.706,Z 650.134,A -85,B 0,C 180,E1 14991.46,E2 14991.46} C_VEL
LIN {X 0,Y 339.702,Z 620.399,A -85,B 0,C 180,E1 14990.248,E2 14990.248} C_VEL
LIN {X 0,Y 339.908,Z 617.912,A -85,B 0,C 180,E1 14990.011,E2 14990.011} C_VEL
LIN {X 0,Y 341.904,Z 608.729,A -85,B 0,C 180,E1 14988.796,E2 14988.796} C_VEL
LIN {X 0,Y 337.762,Z 595.005,A -85,B 0,C 180,E1 14985.756,E2 14985.756} C_VEL
LIN {X 0,Y 333.215,Z 582.164,A -85,B 0,C 180,E1 14982.465,E2 14982.465} C_VEL
LIN {X 0,Y 329.087,Z 571.966,A -85,B 0,C 180,E1 14979.42,E2 14979.42} C_VEL
LIN {X 0,Y 324.867,Z 561.954,A -85,B 0,C 180,E1 14975.968,E2 14975.968} C_VEL
LIN {X 0,Y 320.788,Z 553.327,A -85,B 0,C 180,E1 14972.375,E2 14972.375} C_VEL
LIN {X 0,Y 318.297,Z 548.434,A -85,B 0,C 180,E1 14969.964,E2 14969.964} C_VEL
LIN {X 0,Y 316.101,Z 543.987,A -85,B 0,C 180,E1 14967.504,E2 14967.504} C_VEL
LIN {X 0,Y 314.15,Z 539.895,A -85,B 0,C 180,E1 14964.842,E2 14964.842} C_VEL
LIN {X 0,Y 314.113,Z 539.66,A -85,B 0,C 180,E1 14960.886,E2 14960.886} C_VEL
LIN {X 0,Y 314.106,Z 539.667,A -85,B 0,C 180,E1 14956.457,E2 14956.457} C_VEL
LIN {X 0,Y 314.105,Z 539.672,A -85,B 0,C 180,E1 14952.127,E2 14952.127} C_VEL
LIN {X 0,Y 314.117,Z 539.66,A -85,B 0,C 180,E1 14947.682,E2 14947.682} C_VEL
LIN {X 0,Y 314.133,Z 539.647,A -85,B 0,C 180,E1 14943.284,E2 14943.284} C_VEL
LIN {X 0,Y 314.145,Z 539.641,A -85,B 0,C 180,E1 14938.905,E2 14938.905} C_VEL
LIN {X 0,Y 314.133,Z 539.642,A -85,B 0,C 180,E1 14934.52,E2 14934.52} C_VEL
LIN {X 0,Y 314.161,Z 539.88,A -85,B 0,C 180,E1 14930.196,E2 14930.196} C_VEL
LIN {X 0,Y 316.548,Z 545.185,A -85,B 0,C 180,E1 14926.668,E2 14926.668} C_VEL
LIN {X 0,Y 318.562,Z 549.629,A -85,B 0,C 180,E1 14924.153,E2 14924.153} C_VEL
LIN {X 0,Y 320.407,Z 553.864,A -85,B 0,C 180,E1 14922.004,E2 14922.004} C_VEL
LIN {X 0,Y 323.288,Z 560.502,A -85,B 0,C 180,E1 14918.975,E2 14918.975} C_VEL
LIN {X 0,Y 326.889,Z 570.039,A -85,B 0,C 180,E1 14915.225,E2 14915.225} C_VEL
LIN {X 0,Y 330.414,Z 580.634,A -85,B 0,C 180,E1 14911.634,E2 14911.634} C_VEL
LIN {X 0,Y 333.696,Z 592.22,A -85,B 0,C 180,E1 14908.173,E2 14908.173} C_VEL
LIN {X 0,Y 336.353,Z 603.962,A -85,B 0,C 180,E1 14905.046,E2 14905.046} C_VEL
LIN {X 0,Y 331.45,Z 628.564,A -85,B 0,C 180,E1 14900.568,E2 14900.568} C_VEL
LIN {X 0,Y 337.028,Z 656.944,A -85,B 0,C 180,E1 14898.919,E2 14898.919} C_VEL
LIN {X 0,Y 339.28,Z 671.934,A -85,B 0,C 180,E1 14898.201,E2 14898.201} C_VEL
LIN {X 0,Y 335.597,Z 761.574,A -85,B 0,C 180,E1 14896.096,E2 14896.096} C_VEL
LIN {X 0,Y 334.562,Z 777.559,A -85,B 0,C 180,E1 14895.419,E2 14895.419} C_VEL
LIN {X 0,Y 333.082,Z 792.395,A -85,B 0,C 180,E1 14894.494,E2 14894.494} C_VEL
LIN {X 0,Y 331.098,Z 806.785,A -85,B 0,C 180,E1 14893.267,E2 14893.267} C_VEL
LIN {X 0,Y 328.773,Z 820.429,A -85,B 0,C 180,E1 14891.753,E2 14891.753} C_VEL
LIN {X 0,Y 326.263,Z 832.728,A -85,B 0,C 180,E1 14889.99,E2 14889.99} C_VEL
LIN {X 0,Y 323.703,Z 844.085,A -85,B 0,C 180,E1 14887.922,E2 14887.922} C_VEL
LIN {X 0,Y 321.199,Z 853.98,A -85,B 0,C 180,E1 14885.593,E2 14885.593} C_VEL
LIN {X 0,Y 319.096,Z 861.84,A -85,B 0,C 180,E1 14883.214,E2 14883.214} C_VEL
LIN {X 0,Y 317.202,Z 868.506,A -85,B 0,C 180,E1 14880.491,E2 14880.491} C_VEL
LIN {X 0,Y 315.826,Z 873.283,A -85,B 0,C 180,E1 14877.73,E2 14877.73} C_VEL
LIN {X 0,Y 314.835,Z 876.392,A -85,B 0,C 180,E1 14874.729,E2 14874.729} C_VEL
LIN {X 0,Y 314.314,Z 877.594,A -85,B 0,C 180,E1 14871.846,E2 14871.846} C_VEL
LIN {X 0,Y 314.141,Z 876.958,A -85,B 0,C 180,E1 14868.748,E2 14868.748} C_VEL
LIN {X 0,Y 314.328,Z 874.58,A -85,B 0,C 180,E1 14865.873,E2 14865.873} C_VEL
LIN {X 0,Y 314.903,Z 870.203,A -85,B 0,C 180,E1 14862.897,E2 14862.897} C_VEL
LIN {X 0,Y 315.848,Z 864.015,A -85,B 0,C 180,E1 14860.094,E2 14860.094} C_VEL
LIN {X 0,Y 317.094,Z 856.645,A -85,B 0,C 180,E1 14857.607,E2 14857.607} C_VEL
LIN {X 0,Y 318.671,Z 847.385,A -85,B 0,C 180,E1 14855.218,E2 14855.218} C_VEL
LIN {X 0,Y 320.457,Z 836.647,A -85,B 0,C 180,E1 14853.038,E2 14853.038} C_VEL
LIN {X 0,Y 322.401,Z 823.88,A -85,B 0,C 180,E1 14851.014,E2 14851.014} C_VEL
LIN {X 0,Y 324.203,Z 810.612,A -85,B 0,C 180,E1 14849.379,E2 14849.379} C_VEL
LIN {X 0,Y 325.882,Z 795.852,A -85,B 0,C 180,E1 14847.976,E2 14847.976} C_VEL
LIN {X 0,Y 327.222,Z 780.201,A -85,B 0,C 180,E1 14846.889,E2 14846.889} C_VEL
LIN {X 0,Y 328.127,Z 764.506,A -85,B 0,C 180,E1 14846.138,E2 14846.138} C_VEL
LIN {X 0,Y 328.804,Z 742.387,A -85,B 0,C 180,E1 14845.532,E2 14845.532} C_VEL
LIN {X 0,Y 330.986,Z 666.85,A -85,B 0,C 180,E1 14843.821,E2 14843.821} C_VEL
LIN {X 0,Y 324.928,Z 628.556,A -85,B 0,C 180,E1 14842.261,E2 14842.261} C_VEL
LIN {X 0,Y 328.963,Z 601.6,A -85,B 0,C 180,E1 14837.537,E2 14837.537} C_VEL
LIN {X 0,Y 330.208,Z 593.808,A -85,B 0,C 180,E1 14836.159,E2 14836.159} C_VEL
LIN {X 0,Y 326.52,Z 578.782,A -85,B 0,C 180,E1 14832.72,E2 14832.72} C_VEL
LIN {X 0,Y 323.813,Z 569.083,A -85,B 0,C 180,E1 14830.363,E2 14830.363} C_VEL
LIN {X 0,Y 322.089,Z 565.668,A -85,B 0,C 180,E1 14829.398,E2 14829.398} C_VEL
LIN {X 0,Y 317.348,Z 561.3,A -85,B 0,C 180,E1 14827.759,E2 14827.759} C_VEL
LIN {X 0,Y 312.213,Z 556.581,A -85,B 0,C 180,E1 14825.893,E2 14825.893} C_VEL
LIN {X 0,Y 310.832,Z 553.826,A -85,B 0,C 180,E1 14825.033,E2 14825.033} C_VEL
LIN {X 0,Y 306.906,Z 543.125,A -85,B 0,C 180,E1 14821.811,E2 14821.811} C_VEL
LIN {X 0,Y 306.214,Z 540.752,A -85,B 0,C 180,E1 14821.006,E2 14821.006} C_VEL
LIN {X 0,Y 306.183,Z 540.617,A -85,B 0,C 180,E1 14816.719,E2 14816.719} C_VEL
LIN {X 0,Y 306.171,Z 540.637,A -85,B 0,C 180,E1 14812.214,E2 14812.214} C_VEL
LIN {X 0,Y 306.164,Z 540.631,A -85,B 0,C 180,E1 14807.845,E2 14807.845} C_VEL
LIN {X 0,Y 306.17,Z 540.648,A -85,B 0,C 180,E1 14803.262,E2 14803.262} C_VEL
LIN {X 0,Y 306.183,Z 540.65,A -85,B 0,C 180,E1 14798.829,E2 14798.829} C_VEL
LIN {X 0,Y 306.199,Z 540.614,A -85,B 0,C 180,E1 14794.299,E2 14794.299} C_VEL
LIN {X 0,Y 306.198,Z 540.655,A -85,B 0,C 180,E1 14789.759,E2 14789.759} C_VEL
LIN {X 0,Y 306.179,Z 540.614,A -85,B 0,C 180,E1 14785.328,E2 14785.328} C_VEL
LIN {X 0,Y 306.179,Z 540.655,A -85,B 0,C 180,E1 14780.852,E2 14780.852} C_VEL
LIN {X 0,Y 306.18,Z 540.616,A -85,B 0,C 180,E1 14776.311,E2 14776.311} C_VEL
LIN {X 0,Y 306.2,Z 540.645,A -85,B 0,C 180,E1 14771.872,E2 14771.872} C_VEL
LIN {X 0,Y 306.222,Z 540.612,A -85,B 0,C 180,E1 14767.316,E2 14767.316} C_VEL
LIN {X 0,Y 306.198,Z 540.639,A -85,B 0,C 180,E1 14762.808,E2 14762.808} C_VEL
LIN {X 0,Y 306.188,Z 540.63,A -85,B 0,C 180,E1 14758.316,E2 14758.316} C_VEL
LIN {X 0,Y 306.187,Z 540.626,A -85,B 0,C 180,E1 14753.814,E2 14753.814} C_VEL
LIN {X 0,Y 306.207,Z 540.652,A -85,B 0,C 180,E1 14749.274,E2 14749.274} C_VEL
LIN {X 0,Y 306.226,Z 540.617,A -85,B 0,C 180,E1 14744.859,E2 14744.859} C_VEL
LIN {X 0,Y 306.221,Z 540.636,A -85,B 0,C 180,E1 14740.348,E2 14740.348} C_VEL
LIN {X 0,Y 306.211,Z 540.655,A -85,B 0,C 180,E1 14735.911,E2 14735.911} C_VEL
LIN {X 0,Y 306.201,Z 540.655,A -85,B 0,C 180,E1 14731.314,E2 14731.314} C_VEL
LIN {X 0,Y 306.211,Z 540.654,A -85,B 0,C 180,E1 14726.732,E2 14726.732} C_VEL
LIN {X 0,Y 306.257,Z 540.908,A -85,B 0,C 180,E1 14724.407,E2 14724.407} C_VEL
LIN {X 0,Y 311.66,Z 554.318,A -85,B 0,C 180,E1 14720.802,E2 14720.802} C_VEL
LIN {X 0,Y 317.492,Z 569.745,A -85,B 0,C 180,E1 14717.138,E2 14717.138} C_VEL
LIN {X 0,Y 323.496,Z 587.462,A -85,B 0,C 180,E1 14713.42,E2 14713.42} C_VEL
LIN {X 0,Y 328.625,Z 604.227,A -85,B 0,C 180,E1 14710.248,E2 14710.248} C_VEL
LIN {X 0,Y 326.022,Z 619.014,A -85,B 0,C 180,E1 14708.393,E2 14708.393} C_VEL
LIN {X 0,Y 328.879,Z 652.864,A -85,B 0,C 180,E1 14707.279,E2 14707.279} C_VEL
LIN {X 0,Y 324.239,Z 807.852,A -85,B 0,C 180,E1 14703.954,E2 14703.954} C_VEL
LIN {X 0,Y 322.899,Z 826.24,A -85,B 0,C 180,E1 14703.259,E2 14703.259} C_VEL
LIN {X 0,Y 320.921,Z 844.421,A -85,B 0,C 180,E1 14702.245,E2 14702.245} C_VEL
LIN {X 0,Y 318.684,Z 861.266,A -85,B 0,C 180,E1 14700.966,E2 14700.966} C_VEL
LIN {X 0,Y 316.203,Z 877.769,A -85,B 0,C 180,E1 14699.348,E2 14699.348} C_VEL
LIN {X 0,Y 313.628,Z 893.31,A -85,B 0,C 180,E1 14697.43,E2 14697.43} C_VEL
LIN {X 0,Y 311.136,Z 907.814,A -85,B 0,C 180,E1 14695.201,E2 14695.201} C_VEL
LIN {X 0,Y 308.91,Z 921.275,A -85,B 0,C 180,E1 14692.655,E2 14692.655} C_VEL
LIN {X 0,Y 307.017,Z 933.738,A -85,B 0,C 180,E1 14689.749,E2 14689.749} C_VEL
LIN {X 0,Y 305.757,Z 944.203,A -85,B 0,C 180,E1 14686.725,E2 14686.725} C_VEL
LIN {X 0,Y 305.097,Z 952.704,A -85,B 0,C 180,E1 14683.649,E2 14683.649} C_VEL
LIN {X 0,Y 304.979,Z 959.7,A -85,B 0,C 180,E1 14680.39,E2 14680.39} C_VEL
LIN {X 0,Y 305.246,Z 964.777,A -85,B 0,C 180,E1 14677.152,E2 14677.152} C_VEL
LIN {X 0,Y 305.673,Z 968.074,A -85,B 0,C 180,E1 14673.941,E2 14673.941} C_VEL
LIN {X 0,Y 305.914,Z 969.581,A -85,B 0,C 180,E1 14670.939,E2 14670.939} C_VEL
LIN {X 0,Y 305.825,Z 969.581,A -85,B 0,C 180,E1 14668.129,E2 14668.129} C_VEL
LIN {X 0,Y 305.438,Z 968.155,A -85,B 0,C 180,E1 14665.12,E2 14665.12} C_VEL
LIN {X 0,Y 304.981,Z 965.034,A -85,B 0,C 180,E1 14661.899,E2 14661.899} C_VEL
LIN {X 0,Y 304.792,Z 959.911,A -85,B 0,C 180,E1 14658.46,E2 14658.46} C_VEL
LIN {X 0,Y 305.188,Z 952.833,A -85,B 0,C 180,E1 14655.004,E2 14655.004} C_VEL
LIN {X 0,Y 306.28,Z 944.188,A -85,B 0,C 180,E1 14651.74,E2 14651.74} C_VEL
LIN {X 0,Y 308.084,Z 933.948,A -85,B 0,C 180,E1 14648.659,E2 14648.659} C_VEL
LIN {X 0,Y 310.457,Z 922.434,A -85,B 0,C 180,E1 14645.862,E2 14645.862} C_VEL
LIN {X 0,Y 313.323,Z 909.317,A -85,B 0,C 180,E1 14643.264,E2 14643.264} C_VEL
LIN {X 0,Y 316.49,Z 895.239,A -85,B 0,C 180,E1 14640.997,E2 14640.997} C_VEL
LIN {X 0,Y 319.877,Z 879.507,A -85,B 0,C 180,E1 14638.958,E2 14638.958} C_VEL
LIN {X 0,Y 323.004,Z 863.587,A -85,B 0,C 180,E1 14637.322,E2 14637.322} C_VEL
LIN {X 0,Y 325.968,Z 846.558,A -85,B 0,C 180,E1 14635.965,E2 14635.965} C_VEL
LIN {X 0,Y 328.499,Z 828.784,A -85,B 0,C 180,E1 14634.921,E2 14634.921} C_VEL
LIN {X 0,Y 330.336,Z 810.56,A -85,B 0,C 180,E1 14634.184,E2 14634.184} C_VEL
LIN {X 0,Y 331.403,Z 788.543,A -85,B 0,C 180,E1 14633.634,E2 14633.634} C_VEL
LIN {X 0,Y 336.391,Z 651.075,A -85,B 0,C 180,E1 14630.641,E2 14630.641} C_VEL
LIN {X 0,Y 333.498,Z 621.552,A -85,B 0,C 180,E1 14629.397,E2 14629.397} C_VEL
LIN {X 0,Y 333.348,Z 619.275,A -85,B 0,C 180,E1 14629.263,E2 14629.263} C_VEL
LIN {X 0,Y 335.034,Z 611.794,A -85,B 0,C 180,E1 14628.252,E2 14628.252} C_VEL
LIN {X 0,Y 330.951,Z 598.083,A -85,B 0,C 180,E1 14625.11,E2 14625.11} C_VEL
LIN {X 0,Y 326.642,Z 585.886,A -85,B 0,C 180,E1 14621.859,E2 14621.859} C_VEL
LIN {X 0,Y 322.179,Z 574.643,A -85,B 0,C 180,E1 14618.366,E2 14618.366} C_VEL
LIN {X 0,Y 318.25,Z 565.828,A -85,B 0,C 180,E1 14615.095,E2 14615.095} C_VEL
LIN {X 0,Y 315.122,Z 558.847,A -85,B 0,C 180,E1 14612.107,E2 14612.107} C_VEL
LIN {X 0,Y 312.738,Z 554.071,A -85,B 0,C 180,E1 14609.706,E2 14609.706} C_VEL
LIN {X 0,Y 310.757,Z 549.914,A -85,B 0,C 180,E1 14607.388,E2 14607.388} C_VEL
LIN {X 0,Y 308.257,Z 545.1,A -85,B 0,C 180,E1 14604.122,E2 14604.122} C_VEL
LIN {X 0,Y 306.196,Z 540.794,A -85,B 0,C 180,E1 14600.36,E2 14600.36} C_VEL
LIN {X 0,Y 306.181,Z 540.641,A -85,B 0,C 180,E1 14595.92,E2 14595.92} C_VEL
LIN {X 0,Y 306.19,Z 540.649,A -85,B 0,C 180,E1 14591.49,E2 14591.49} C_VEL
LIN {X 0,Y 306.187,Z 540.659,A -85,B 0,C 180,E1 14586.939,E2 14586.939} C_VEL
LIN {X 0,Y 306.175,Z 540.655,A -85,B 0,C 180,E1 14582.433,E2 14582.433} C_VEL
LIN {X 0,Y 306.178,Z 540.651,A -85,B 0,C 180,E1 14577.754,E2 14577.754} C_VEL
LIN {X 0,Y 306.232,Z 540.947,A -85,B 0,C 180,E1 14574.378,E2 14574.378} C_VEL
LIN {X 0,Y 308.609,Z 545.888,A -85,B 0,C 180,E1 14570.112,E2 14570.112} C_VEL
LIN {X 0,Y 310.76,Z 550.441,A -85,B 0,C 180,E1 14566.984,E2 14566.984} C_VEL
LIN {X 0,Y 312.81,Z 555.244,A -85,B 0,C 180,E1 14564.235,E2 14564.235} C_VEL
LIN {X 0,Y 314.604,Z 559.478,A -85,B 0,C 180,E1 14562.044,E2 14562.044} C_VEL
LIN {X 0,Y 317.245,Z 565.708,A -85,B 0,C 180,E1 14559.136,E2 14559.136} C_VEL
LIN {X 0,Y 320.604,Z 574.757,A -85,B 0,C 180,E1 14555.494,E2 14555.494} C_VEL
LIN {X 0,Y 324.011,Z 585.314,A -85,B 0,C 180,E1 14551.826,E2 14551.826} C_VEL
LIN {X 0,Y 327.194,Z 596.946,A -85,B 0,C 180,E1 14548.29,E2 14548.29} C_VEL
LIN {X 0,Y 329.389,Z 607.342,A -85,B 0,C 180,E1 14545.467,E2 14545.467} C_VEL
LIN {X 0,Y 324.963,Z 628.487,A -85,B 0,C 180,E1 14541.572,E2 14541.572} C_VEL
LIN {X 0,Y 330.248,Z 655.35,A -85,B 0,C 180,E1 14539.928,E2 14539.928} C_VEL
LIN {X 0,Y 332.97,Z 673.044,A -85,B 0,C 180,E1 14539.027,E2 14539.027} C_VEL
LIN {X 0,Y 329.108,Z 762.266,A -85,B 0,C 180,E1 14536.894,E2 14536.894} C_VEL
LIN {X 0,Y 328.007,Z 778.358,A -85,B 0,C 180,E1 14536.2,E2 14536.2} C_VEL
LIN {X 0,Y 326.344,Z 794.06,A -85,B 0,C 180,E1 14535.196,E2 14535.196} C_VEL
LIN {X 0,Y 324.227,Z 808.448,A -85,B 0,C 180,E1 14533.929,E2 14533.929} C_VEL
LIN {X 0,Y 321.79,Z 821.926,A -85,B 0,C 180,E1 14532.389,E2 14532.389} C_VEL
LIN {X 0,Y 319.036,Z 834.641,A -85,B 0,C 180,E1 14530.507,E2 14530.507} C_VEL
LIN {X 0,Y 316.459,Z 845.389,A -85,B 0,C 180,E1 14528.487,E2 14528.487} C_VEL
LIN {X 0,Y 313.815,Z 855.235,A -85,B 0,C 180,E1 14526.111,E2 14526.111} C_VEL
LIN {X 0,Y 311.608,Z 862.973,A -85,B 0,C 180,E1 14523.712,E2 14523.712} C_VEL
LIN {X 0,Y 309.56,Z 869.708,A -85,B 0,C 180,E1 14520.896,E2 14520.896} C_VEL
LIN {X 0,Y 308.054,Z 874.541,A -85,B 0,C 180,E1 14518.012,E2 14518.012} C_VEL
LIN {X 0,Y 306.963,Z 877.687,A -85,B 0,C 180,E1 14514.842,E2 14514.842} C_VEL
LIN {X 0,Y 306.401,Z 878.794,A -85,B 0,C 180,E1 14511.835,E2 14511.835} C_VEL
LIN {X 0,Y 306.226,Z 878.079,A -85,B 0,C 180,E1 14508.658,E2 14508.658} C_VEL
LIN {X 0,Y 306.428,Z 875.596,A -85,B 0,C 180,E1 14505.71,E2 14505.71} C_VEL
LIN {X 0,Y 307.008,Z 871.376,A -85,B 0,C 180,E1 14502.791,E2 14502.791} C_VEL
LIN {X 0,Y 307.998,Z 865.166,A -85,B 0,C 180,E1 14499.904,E2 14499.904} C_VEL
LIN {X 0,Y 309.256,Z 858.042,A -85,B 0,C 180,E1 14497.428,E2 14497.428} C_VEL
LIN {X 0,Y 310.889,Z 848.872,A -85,B 0,C 180,E1 14494.979,E2 14494.979} C_VEL
LIN {X 0,Y 312.741,Z 838.269,A -85,B 0,C 180,E1 14492.746,E2 14492.746} C_VEL
LIN {X 0,Y 314.696,Z 825.988,A -85,B 0,C 180,E1 14490.726,E2 14490.726} C_VEL
LIN {X 0,Y 316.515,Z 813.453,A -85,B 0,C 180,E1 14489.093,E2 14489.093} C_VEL
LIN {X 0,Y 318.242,Z 799.18,A -85,B 0,C 180,E1 14487.657,E2 14487.657} C_VEL
LIN {X 0,Y 319.647,Z 784.6,A -85,B 0,C 180,E1 14486.546,E2 14486.546} C_VEL
LIN {X 0,Y 320.758,Z 767.682,A -85,B 0,C 180,E1 14485.652,E2 14485.652} C_VEL
LIN {X 0,Y 321.359,Z 750.352,A -85,B 0,C 180,E1 14485.107,E2 14485.107} C_VEL
LIN {X 0,Y 323.851,Z 667.924,A -85,B 0,C 180,E1 14483.2,E2 14483.2} C_VEL
LIN {X 0,Y 317.665,Z 628.711,A -85,B 0,C 180,E1 14481.582,E2 14481.582} C_VEL
LIN {X 0,Y 321.786,Z 602.334,A -85,B 0,C 180,E1 14476.889,E2 14476.889} C_VEL
LIN {X 0,Y 322.75,Z 596.012,A -85,B 0,C 180,E1 14475.741,E2 14475.741} C_VEL
LIN {X 0,Y 318.939,Z 580.559,A -85,B 0,C 180,E1 14472.107,E2 14472.107} C_VEL
LIN {X 0,Y 314.643,Z 565.487,A -85,B 0,C 180,E1 14468.271,E2 14468.271} C_VEL
LIN {X 0,Y 310.832,Z 553.826,A -85,B 0,C 180,E1 14465.033,E2 14465.033} C_VEL
LIN {X 0,Y 309.425,Z 551.877,A -85,B 0,C 180,E1 14464.337,E2 14464.337} C_VEL
LIN {X 0,Y 304.925,Z 549.917,A -85,B 0,C 180,E1 14463.07,E2 14463.07} C_VEL
LIN {X 0,Y 300.946,Z 548.037,A -85,B 0,C 180,E1 14461.888,E2 14461.888} C_VEL
LIN {X 0,Y 299.855,Z 546.398,A -85,B 0,C 180,E1 14461.277,E2 14461.277} C_VEL
LIN {X 0,Y 298.243,Z 541.76,A -85,B 0,C 180,E1 14459.699,E2 14459.699} C_VEL
LIN {X 0,Y 298.242,Z 541.649,A -85,B 0,C 180,E1 14455.223,E2 14455.223} C_VEL
LIN {X 0,Y 298.269,Z 541.641,A -85,B 0,C 180,E1 14450.687,E2 14450.687} C_VEL
LIN {X 0,Y 298.24,Z 541.624,A -85,B 0,C 180,E1 14446.121,E2 14446.121} C_VEL
LIN {X 0,Y 298.227,Z 541.613,A -85,B 0,C 180,E1 14441.593,E2 14441.593} C_VEL
LIN {X 0,Y 298.235,Z 541.647,A -85,B 0,C 180,E1 14437.071,E2 14437.071} C_VEL
LIN {X 0,Y 298.255,Z 541.616,A -85,B 0,C 180,E1 14432.438,E2 14432.438} C_VEL
LIN {X 0,Y 298.27,Z 541.616,A -85,B 0,C 180,E1 14427.99,E2 14427.99} C_VEL
LIN {X 0,Y 298.256,Z 541.629,A -85,B 0,C 180,E1 14423.512,E2 14423.512} C_VEL
LIN {X 0,Y 298.242,Z 541.607,A -85,B 0,C 180,E1 14419.027,E2 14419.027} C_VEL
LIN {X 0,Y 298.246,Z 541.64,A -85,B 0,C 180,E1 14414.346,E2 14414.346} C_VEL
LIN {X 0,Y 298.26,Z 541.595,A -85,B 0,C 180,E1 14409.758,E2 14409.758} C_VEL
LIN {X 0,Y 298.276,Z 541.635,A -85,B 0,C 180,E1 14405.386,E2 14405.386} C_VEL
LIN {X 0,Y 298.259,Z 541.593,A -85,B 0,C 180,E1 14400.769,E2 14400.769} C_VEL
LIN {X 0,Y 298.255,Z 541.645,A -85,B 0,C 180,E1 14396.348,E2 14396.348} C_VEL
LIN {X 0,Y 298.25,Z 541.604,A -85,B 0,C 180,E1 14391.712,E2 14391.712} C_VEL
LIN {X 0,Y 298.267,Z 541.629,A -85,B 0,C 180,E1 14387.218,E2 14387.218} C_VEL
LIN {X 0,Y 298.287,Z 541.637,A -85,B 0,C 180,E1 14382.643,E2 14382.643} C_VEL
LIN {X 0,Y 298.278,Z 541.614,A -85,B 0,C 180,E1 14378.156,E2 14378.156} C_VEL
LIN {X 0,Y 298.267,Z 541.618,A -85,B 0,C 180,E1 14373.737,E2 14373.737} C_VEL
LIN {X 0,Y 298.262,Z 541.624,A -85,B 0,C 180,E1 14369.11,E2 14369.11} C_VEL
LIN {X 0,Y 298.322,Z 541.928,A -85,B 0,C 180,E1 14365.77,E2 14365.77} C_VEL
LIN {X 0,Y 303.369,Z 554.479,A -85,B 0,C 180,E1 14362.192,E2 14362.192} C_VEL
LIN {X 0,Y 308.83,Z 568.438,A -85,B 0,C 180,E1 14358.665,E2 14358.665} C_VEL
LIN {X 0,Y 314.709,Z 585.348,A -85,B 0,C 180,E1 14354.888,E2 14354.888} C_VEL
LIN {X 0,Y 320.425,Z 603.689,A -85,B 0,C 180,E1 14351.235,E2 14351.235} C_VEL
LIN {X 0,Y 321.261,Z 606.526,A -85,B 0,C 180,E1 14350.705,E2 14350.705} C_VEL
LIN {X 0,Y 318.953,Z 619.227,A -85,B 0,C 180,E1 14349.083,E2 14349.083} C_VEL
LIN {X 0,Y 321.776,Z 653.686,A -85,B 0,C 180,E1 14347.92,E2 14347.92} C_VEL
LIN {X 0,Y 316.99,Z 807.266,A -85,B 0,C 180,E1 14344.566,E2 14344.566} C_VEL
LIN {X 0,Y 315.613,Z 825.646,A -85,B 0,C 180,E1 14343.858,E2 14343.858} C_VEL
LIN {X 0,Y 313.574,Z 843.832,A -85,B 0,C 180,E1 14342.823,E2 14342.823} C_VEL
LIN {X 0,Y 311.182,Z 861.19,A -85,B 0,C 180,E1 14341.475,E2 14341.475} C_VEL
LIN {X 0,Y 308.618,Z 877.55,A -85,B 0,C 180,E1 14339.822,E2 14339.822} C_VEL
LIN {X 0,Y 305.958,Z 892.926,A -85,B 0,C 180,E1 14337.86,E2 14337.86} C_VEL
LIN {X 0,Y 303.374,Z 907.325,A -85,B 0,C 180,E1 14335.579,E2 14335.579} C_VEL
LIN {X 0,Y 301.145,Z 920.253,A -85,B 0,C 180,E1 14333.066,E2 14333.066} C_VEL
LIN {X 0,Y 299.163,Z 932.694,A -85,B 0,C 180,E1 14330.09,E2 14330.09} C_VEL
LIN {X 0,Y 297.837,Z 943.165,A -85,B 0,C 180,E1 14326.983,E2 14326.983} C_VEL
LIN {X 0,Y 297.143,Z 951.654,A -85,B 0,C 180,E1 14323.823,E2 14323.823} C_VEL
LIN {X 0,Y 297.02,Z 958.628,A -85,B 0,C 180,E1 14320.475,E2 14320.475} C_VEL
LIN {X 0,Y 297.309,Z 963.682,A -85,B 0,C 180,E1 14317.15,E2 14317.15} C_VEL
LIN {X 0,Y 297.739,Z 966.815,A -85,B 0,C 180,E1 14314.046,E2 14314.046} C_VEL
LIN {X 0,Y 298.005,Z 968.36,A -85,B 0,C 180,E1 14310.963,E2 14310.963} C_VEL
LIN {X 0,Y 297.903,Z 968.401,A -85,B 0,C 180,E1 14308.079,E2 14308.079} C_VEL
LIN {X 0,Y 297.479,Z 967.007,A -85,B 0,C 180,E1 14304.989,E2 14304.989} C_VEL
LIN {X 0,Y 296.995,Z 963.916,A -85,B 0,C 180,E1 14301.68,E2 14301.68} C_VEL
LIN {X 0,Y 296.816,Z 958.816,A -85,B 0,C 180,E1 14298.146,E2 14298.146} C_VEL
LIN {X 0,Y 297.279,Z 951.76,A -85,B 0,C 180,E1 14294.595,E2 14294.595} C_VEL
LIN {X 0,Y 298.481,Z 943.138,A -85,B 0,C 180,E1 14291.245,E2 14291.245} C_VEL
LIN {X 0,Y 300.408,Z 933.041,A -85,B 0,C 180,E1 14288.118,E2 14288.118} C_VEL
LIN {X 0,Y 303.071,Z 921.039,A -85,B 0,C 180,E1 14285.128,E2 14285.128} C_VEL
LIN {X 0,Y 306.145,Z 907.905,A -85,B 0,C 180,E1 14282.48,E2 14282.48} C_VEL
LIN {X 0,Y 309.666,Z 893.133,A -85,B 0,C 180,E1 14280.081,E2 14280.081} C_VEL
LIN {X 0,Y 313.092,Z 877.919,A -85,B 0,C 180,E1 14278.1,E2 14278.1} C_VEL
LIN {X 0,Y 316.412,Z 861.765,A -85,B 0,C 180,E1 14276.433,E2 14276.433} C_VEL
LIN {X 0,Y 319.511,Z 844.538,A -85,B 0,C 180,E1 14275.07,E2 14275.07} C_VEL
LIN {X 0,Y 322.069,Z 826.885,A -85,B 0,C 180,E1 14274.045,E2 14274.045} C_VEL
LIN {X 0,Y 323.924,Z 808.682,A -85,B 0,C 180,E1 14273.317,E2 14273.317} C_VEL
LIN {X 0,Y 325.141,Z 782.72,A -85,B 0,C 180,E1 14272.685,E2 14272.685} C_VEL
LIN {X 0,Y 330.184,Z 651.974,A -85,B 0,C 180,E1 14269.78,E2 14269.78} C_VEL
LIN {X 0,Y 327.386,Z 622.602,A -85,B 0,C 180,E1 14268.502,E2 14268.502} C_VEL
LIN {X 0,Y 327.142,Z 619.454,A -85,B 0,C 180,E1 14268.323,E2 14268.323} C_VEL
LIN {X 0,Y 328.185,Z 614.839,A -85,B 0,C 180,E1 14267.685,E2 14267.685} C_VEL
LIN {X 0,Y 324.385,Z 601.875,A -85,B 0,C 180,E1 14264.609,E2 14264.609} C_VEL
LIN {X 0,Y 320.097,Z 589.629,A -85,B 0,C 180,E1 14261.23,E2 14261.23} C_VEL
LIN {X 0,Y 315.97,Z 579.242,A -85,B 0,C 180,E1 14257.871,E2 14257.871} C_VEL
LIN {X 0,Y 312.287,Z 570.729,A -85,B 0,C 180,E1 14254.641,E2 14254.641} C_VEL
LIN {X 0,Y 309.404,Z 564.267,A -85,B 0,C 180,E1 14251.785,E2 14251.785} C_VEL
LIN {X 0,Y 307.185,Z 559.701,A -85,B 0,C 180,E1 14249.438,E2 14249.438} C_VEL
LIN {X 0,Y 305.218,Z 555.603,A -85,B 0,C 180,E1 14247.087,E2 14247.087} C_VEL
LIN {X 0,Y 302.911,Z 550.987,A -85,B 0,C 180,E1 14243.906,E2 14243.906} C_VEL
LIN {X 0,Y 300.559,Z 546.356,A -85,B 0,C 180,E1 14239.835,E2 14239.835} C_VEL
LIN {X 0,Y 298.278,Z 541.84,A -85,B 0,C 180,E1 14233.176,E2 14233.176} C_VEL
LIN {X 0,Y 298.223,Z 541.624,A -85,B 0,C 180,E1 14228.535,E2 14228.535} C_VEL
LIN {X 0,Y 298.236,Z 541.658,A -85,B 0,C 180,E1 14223.844,E2 14223.844} C_VEL
LIN {X 0,Y 298.363,Z 542.228,A -85,B 0,C 180,E1 14220.96,E2 14220.96} C_VEL
LIN {X 0,Y 300.774,Z 546.81,A -85,B 0,C 180,E1 14214.467,E2 14214.467} C_VEL
LIN {X 0,Y 303.093,Z 551.811,A -85,B 0,C 180,E1 14210.122,E2 14210.122} C_VEL
LIN {X 0,Y 305.084,Z 556.077,A -85,B 0,C 180,E1 14207.123,E2 14207.123} C_VEL
LIN {X 0,Y 306.958,Z 560.498,A -85,B 0,C 180,E1 14204.508,E2 14204.508} C_VEL
LIN {X 0,Y 308.774,Z 564.952,A -85,B 0,C 180,E1 14202.156,E2 14202.156} C_VEL
LIN {X 0,Y 311.205,Z 570.91,A -85,B 0,C 180,E1 14199.303,E2 14199.303} C_VEL
LIN {X 0,Y 314.483,Z 580.015,A -85,B 0,C 180,E1 14195.586,E2 14195.586} C_VEL
LIN {X 0,Y 317.64,Z 590.032,A -85,B 0,C 180,E1 14192.029,E2 14192.029} C_VEL
LIN {X 0,Y 320.543,Z 601.026,A -85,B 0,C 180,E1 14188.606,E2 14188.606} C_VEL
LIN {X 0,Y 322.52,Z 610.444,A -85,B 0,C 180,E1 14185.973,E2 14185.973} C_VEL
LIN {X 0,Y 318.593,Z 628.018,A -85,B 0,C 180,E1 14182.663,E2 14182.663} C_VEL
LIN {X 0,Y 319.816,Z 634.752,A -85,B 0,C 180,E1 14182.167,E2 14182.167} C_VEL
LIN {X 0,Y 325.393,Z 664.46,A -85,B 0,C 180,E1 14180.386,E2 14180.386} C_VEL
LIN {X 0,Y 326.743,Z 674.544,A -85,B 0,C 180,E1 14179.882,E2 14179.882} C_VEL
LIN {X 0,Y 322.735,Z 762.96,A -85,B 0,C 180,E1 14177.735,E2 14177.735} C_VEL
LIN {X 0,Y 321.578,Z 779.006,A -85,B 0,C 180,E1 14177.033,E2 14177.033} C_VEL
LIN {X 0,Y 319.913,Z 794.033,A -85,B 0,C 180,E1 14176.064,E2 14176.064} C_VEL
LIN {X 0,Y 317.741,Z 808.288,A -85,B 0,C 180,E1 14174.812,E2 14174.812} C_VEL
LIN {X 0,Y 315.162,Z 821.951,A -85,B 0,C 180,E1 14173.249,E2 14173.249} C_VEL
LIN {X 0,Y 312.449,Z 834.01,A -85,B 0,C 180,E1 14171.477,E2 14171.477} C_VEL
LIN {X 0,Y 309.497,Z 845.75,A -85,B 0,C 180,E1 14169.279,E2 14169.279} C_VEL
LIN {X 0,Y 306.86,Z 855.124,A -85,B 0,C 180,E1 14167.031,E2 14167.031} C_VEL
LIN {X 0,Y 304.296,Z 863.609,A -85,B 0,C 180,E1 14164.407,E2 14164.407} C_VEL
LIN {X 0,Y 302.212,Z 870.086,A -85,B 0,C 180,E1 14161.733,E2 14161.733} C_VEL
LIN {X 0,Y 300.438,Z 875.379,A -85,B 0,C 180,E1 14158.63,E2 14158.63} C_VEL
LIN {X 0,Y 299.263,Z 878.553,A -85,B 0,C 180,E1 14155.565,E2 14155.565} C_VEL
LIN {X 0,Y 298.574,Z 879.961,A -85,B 0,C 180,E1 14152.438,E2 14152.438} C_VEL
LIN {X 0,Y 298.312,Z 879.547,A -85,B 0,C 180,E1 14149.375,E2 14149.375} C_VEL
LIN {X 0,Y 298.433,Z 877.468,A -85,B 0,C 180,E1 14146.342,E2 14146.342} C_VEL
LIN {X 0,Y 298.941,Z 873.603,A -85,B 0,C 180,E1 14143.34,E2 14143.34} C_VEL
LIN {X 0,Y 299.878,Z 867.892,A -85,B 0,C 180,E1 14140.369,E2 14140.369} C_VEL
LIN {X 0,Y 301.187,Z 860.584,A -85,B 0,C 180,E1 14137.628,E2 14137.628} C_VEL
LIN {X 0,Y 302.824,Z 851.877,A -85,B 0,C 180,E1 14135.112,E2 14135.112} C_VEL
LIN {X 0,Y 304.674,Z 841.692,A -85,B 0,C 180,E1 14132.819,E2 14132.819} C_VEL
LIN {X 0,Y 306.664,Z 830.11,A -85,B 0,C 180,E1 14130.745,E2 14130.745} C_VEL
LIN {X 0,Y 308.702,Z 816.79,A -85,B 0,C 180,E1 14128.884,E2 14128.884} C_VEL
LIN {X 0,Y 310.497,Z 803.339,A -85,B 0,C 180,E1 14127.414,E2 14127.414} C_VEL
LIN {X 0,Y 312.117,Z 787.821,A -85,B 0,C 180,E1 14126.141,E2 14126.141} C_VEL
LIN {X 0,Y 313.294,Z 772.107,A -85,B 0,C 180,E1 14125.221,E2 14125.221} C_VEL
LIN {X 0,Y 314.036,Z 754.849,A -85,B 0,C 180,E1 14124.589,E2 14124.589} C_VEL
LIN {X 0,Y 316.729,Z 668.925,A -85,B 0,C 180,E1 14122.555,E2 14122.555} C_VEL
LIN {X 0,Y 310.463,Z 628.469,A -85,B 0,C 180,E1 14120.825,E2 14120.825} C_VEL
LIN {X 0,Y 314.817,Z 602.085,A -85,B 0,C 180,E1 14116.031,E2 14116.031} C_VEL
LIN {X 0,Y 315.284,Z 598.221,A -85,B 0,C 180,E1 14115.297,E2 14115.297} C_VEL
LIN {X 0,Y 311.6,Z 583.153,A -85,B 0,C 180,E1 14111.671,E2 14111.671} C_VEL
LIN {X 0,Y 307.457,Z 568.494,A -85,B 0,C 180,E1 14107.837,E2 14107.837} C_VEL
LIN {X 0,Y 303.31,Z 555.812,A -85,B 0,C 180,E1 14104.206,E2 14104.206} C_VEL
LIN {X 0,Y 299.855,Z 546.398,A -85,B 0,C 180,E1 14101.277,E2 14101.277} C_VEL
LIN {X 0,Y 298.219,Z 544.226,A -85,B 0,C 180,E1 14100.41,E2 14100.41} C_VEL
LIN {X 0,Y 294.19,Z 542.825,A -85,B 0,C 180,E1 14099.17,E2 14099.17} C_VEL
LIN {X 0,Y 291.086,Z 542.564,A -85,B 0,C 180,E1 14097.952,E2 14097.952} C_VEL
LIN {X 0,Y 290.305,Z 542.579,A -85,B 0,C 180,E1 14097.065,E2 14097.065} C_VEL
LIN {X 0,Y 290.304,Z 542.611,A -85,B 0,C 180,E1 14092.439,E2 14092.439} C_VEL
LIN {X 0,Y 290.293,Z 542.608,A -85,B 0,C 180,E1 14088.071,E2 14088.071} C_VEL
LIN {X 0,Y 290.291,Z 542.627,A -85,B 0,C 180,E1 14083.387,E2 14083.387} C_VEL
LIN {X 0,Y 290.306,Z 542.626,A -85,B 0,C 180,E1 14078.818,E2 14078.818} C_VEL
LIN {X 0,Y 290.322,Z 542.589,A -85,B 0,C 180,E1 14074.151,E2 14074.151} C_VEL
LIN {X 0,Y 290.307,Z 542.633,A -85,B 0,C 180,E1 14069.506,E2 14069.506} C_VEL
LIN {X 0,Y 290.296,Z 542.595,A -85,B 0,C 180,E1 14064.848,E2 14064.848} C_VEL
LIN {X 0,Y 290.309,Z 542.62,A -85,B 0,C 180,E1 14060.357,E2 14060.357} C_VEL
LIN {X 0,Y 290.33,Z 542.596,A -85,B 0,C 180,E1 14055.788,E2 14055.788} C_VEL
LIN {X 0,Y 290.327,Z 542.611,A -85,B 0,C 180,E1 14051.321,E2 14051.321} C_VEL
LIN {X 0,Y 290.309,Z 542.602,A -85,B 0,C 180,E1 14046.725,E2 14046.725} C_VEL
LIN {X 0,Y 290.305,Z 542.599,A -85,B 0,C 180,E1 14042.172,E2 14042.172} C_VEL
LIN {X 0,Y 290.319,Z 542.621,A -85,B 0,C 180,E1 14037.632,E2 14037.632} C_VEL
LIN {X 0,Y 290.344,Z 542.588,A -85,B 0,C 180,E1 14033.078,E2 14033.078} C_VEL
LIN {X 0,Y 290.334,Z 542.633,A -85,B 0,C 180,E1 14028.479,E2 14028.479} C_VEL
LIN {X 0,Y 290.316,Z 542.607,A -85,B 0,C 180,E1 14023.802,E2 14023.802} C_VEL
LIN {X 0,Y 290.321,Z 542.602,A -85,B 0,C 180,E1 14019.223,E2 14019.223} C_VEL
LIN {X 0,Y 290.337,Z 542.614,A -85,B 0,C 180,E1 14014.721,E2 14014.721} C_VEL
LIN {X 0,Y 290.362,Z 542.62,A -85,B 0,C 180,E1 14010.196,E2 14010.196} C_VEL
LIN {X 0,Y 290.361,Z 542.871,A -85,B 0,C 180,E1 14007.274,E2 14007.274} C_VEL
LIN {X 0,Y 295.11,Z 554.392,A -85,B 0,C 180,E1 14003.74,E2 14003.74} C_VEL
LIN {X 0,Y 300.506,Z 568.18,A -85,B 0,C 180,E1 14000.047,E2 14000.047} C_VEL
LIN {X 0,Y 305.963,Z 583.506,A -85,B 0,C 180,E1 13996.408,E2 13996.408} C_VEL
LIN {X 0,Y 311.545,Z 601.088,A -85,B 0,C 180,E1 13992.698,E2 13992.698} C_VEL
LIN {X 0,Y 313.856,Z 609.035,A -85,B 0,C 180,E1 13991.147,E2 13991.147} C_VEL
LIN {X 0,Y 311.922,Z 619.351,A -85,B 0,C 180,E1 13989.807,E2 13989.807} C_VEL
LIN {X 0,Y 314.716,Z 654.542,A -85,B 0,C 180,E1 13988.59,E2 13988.59} C_VEL
LIN {X 0,Y 309.764,Z 806.588,A -85,B 0,C 180,E1 13985.202,E2 13985.202} C_VEL
LIN {X 0,Y 308.358,Z 824.868,A -85,B 0,C 180,E1 13984.484,E2 13984.484} C_VEL
LIN {X 0,Y 306.259,Z 843.055,A -85,B 0,C 180,E1 13983.43,E2 13983.43} C_VEL
LIN {X 0,Y 303.857,Z 859.877,A -85,B 0,C 180,E1 13982.101,E2 13982.101} C_VEL
LIN {X 0,Y 301.192,Z 876.354,A -85,B 0,C 180,E1 13980.414,E2 13980.414} C_VEL
LIN {X 0,Y 298.427,Z 891.835,A -85,B 0,C 180,E1 13978.409,E2 13978.409} C_VEL
LIN {X 0,Y 295.728,Z 906.282,A -85,B 0,C 180,E1 13976.074,E2 13976.074} C_VEL
LIN {X 0,Y 293.397,Z 919.229,A -85,B 0,C 180,E1 13973.499,E2 13973.499} C_VEL
LIN {X 0,Y 291.323,Z 931.645,A -85,B 0,C 180,E1 13970.451,E2 13970.451} C_VEL
LIN {X 0,Y 289.919,Z 942.127,A -85,B 0,C 180,E1 13967.254,E2 13967.254} C_VEL
LIN {X 0,Y 289.19,Z 950.604,A -85,B 0,C 180,E1 13964.007,E2 13964.007} C_VEL
LIN {X 0,Y 289.06,Z 957.549,A -85,B 0,C 180,E1 13960.565,E2 13960.565} C_VEL
LIN {X 0,Y 289.374,Z 962.58,A -85,B 0,C 180,E1 13957.147,E2 13957.147} C_VEL
LIN {X 0,Y 289.832,Z 965.686,A -85,B 0,C 180,E1 13953.958,E2 13953.958} C_VEL
LIN {X 0,Y 290.101,Z 967.198,A -85,B 0,C 180,E1 13950.792,E2 13950.792} C_VEL
LIN {X 0,Y 289.958,Z 967.184,A -85,B 0,C 180,E1 13947.829,E2 13947.829} C_VEL
LIN {X 0,Y 289.485,Z 965.724,A -85,B 0,C 180,E1 13944.652,E2 13944.652} C_VEL
LIN {X 0,Y 288.967,Z 962.321,A -85,B 0,C 180,E1 13941.046,E2 13941.046} C_VEL
LIN {X 0,Y 288.861,Z 957.042,A -85,B 0,C 180,E1 13937.408,E2 13937.408} C_VEL
LIN {X 0,Y 289.496,Z 949.804,A -85,B 0,C 180,E1 13933.758,E2 13933.758} C_VEL
LIN {X 0,Y 290.916,Z 940.993,A -85,B 0,C 180,E1 13930.321,E2 13930.321} C_VEL
LIN {X 0,Y 293.171,Z 930.375,A -85,B 0,C 180,E1 13927.048,E2 13927.048} C_VEL
LIN {X 0,Y 295.946,Z 918.815,A -85,B 0,C 180,E1 13924.167,E2 13924.167} C_VEL
LIN {X 0,Y 299.287,Z 905.447,A -85,B 0,C 180,E1 13921.468,E2 13921.468} C_VEL
LIN {X 0,Y 302.776,Z 891.647,A -85,B 0,C 180,E1 13919.218,E2 13919.218} C_VEL
LIN {X 0,Y 306.385,Z 876.331,A -85,B 0,C 180,E1 13917.205,E2 13917.205} C_VEL
LIN {X 0,Y 309.892,Z 860.058,A -85,B 0,C 180,E1 13915.517,E2 13915.517} C_VEL
LIN {X 0,Y 312.93,Z 843.856,A -85,B 0,C 180,E1 13914.224,E2 13914.224} C_VEL
LIN {X 0,Y 315.611,Z 826.205,A -85,B 0,C 180,E1 13913.183,E2 13913.183} C_VEL
LIN {X 0,Y 317.536,Z 808.118,A -85,B 0,C 180,E1 13912.447,E2 13912.447} C_VEL
LIN {X 0,Y 318.793,Z 782.82,A -85,B 0,C 180,E1 13911.817,E2 13911.817} C_VEL
LIN {X 0,Y 324.064,Z 652.989,A -85,B 0,C 180,E1 13908.891,E2 13908.891} C_VEL
LIN {X 0,Y 321.349,Z 623.555,A -85,B 0,C 180,E1 13907.569,E2 13907.569} C_VEL
LIN {X 0,Y 321.086,Z 619.381,A -85,B 0,C 180,E1 13907.314,E2 13907.314} C_VEL
LIN {X 0,Y 321.298,Z 617.684,A -85,B 0,C 180,E1 13907.046,E2 13907.046} C_VEL
LIN {X 0,Y 317.517,Z 604.795,A -85,B 0,C 180,E1 13903.85,E2 13903.85} C_VEL
LIN {X 0,Y 313.563,Z 593.432,A -85,B 0,C 180,E1 13900.579,E2 13900.579} C_VEL
LIN {X 0,Y 309.967,Z 584.185,A -85,B 0,C 180,E1 13897.494,E2 13897.494} C_VEL
LIN {X 0,Y 306.007,Z 574.562,A -85,B 0,C 180,E1 13893.742,E2 13893.742} C_VEL
LIN {X 0,Y 303.189,Z 568.717,A -85,B 0,C 180,E1 13890.961,E2 13890.961} C_VEL
LIN {X 0,Y 301.619,Z 565.314,A -85,B 0,C 180,E1 13889.163,E2 13889.163} C_VEL
LIN {X 0,Y 299.876,Z 561.527,A -85,B 0,C 180,E1 13886.965,E2 13886.965} C_VEL
LIN {X 0,Y 297.629,Z 556.963,A -85,B 0,C 180,E1 13883.774,E2 13883.774} C_VEL
LIN {X 0,Y 295.281,Z 552.316,A -85,B 0,C 180,E1 13879.586,E2 13879.586} C_VEL
LIN {X 0,Y 292.976,Z 547.785,A -85,B 0,C 180,E1 13872.816,E2 13872.816} C_VEL
LIN {X 0,Y 292.235,Z 546.909,A -85,B 0,C 180,E1 13867.47,E2 13867.47} C_VEL
LIN {X 0,Y 292.808,Z 547.596,A -85,B 0,C 180,E1 13862.544,E2 13862.544} C_VEL
LIN {X 0,Y 293.504,Z 549.652,A -85,B 0,C 180,E1 13858.828,E2 13858.828} C_VEL
LIN {X 0,Y 295.423,Z 552.956,A -85,B 0,C 180,E1 13854.367,E2 13854.367} C_VEL
LIN {X 0,Y 297.513,Z 557.446,A -85,B 0,C 180,E1 13850.326,E2 13850.326} C_VEL
LIN {X 0,Y 299.507,Z 562.055,A -85,B 0,C 180,E1 13847.075,E2 13847.075} C_VEL
LIN {X 0,Y 301.206,Z 566.096,A -85,B 0,C 180,E1 13844.599,E2 13844.599} C_VEL
LIN {X 0,Y 303.748,Z 572.099,A -85,B 0,C 180,E1 13841.379,E2 13841.379} C_VEL
LIN {X 0,Y 306.918,Z 580.977,A -85,B 0,C 180,E1 13837.392,E2 13837.392} C_VEL
LIN {X 0,Y 310.078,Z 590.657,A -85,B 0,C 180,E1 13833.677,E2 13833.677} C_VEL
LIN {X 0,Y 313.016,Z 601.28,A -85,B 0,C 180,E1 13830.111,E2 13830.111} C_VEL
LIN {X 0,Y 315.505,Z 612.67,A -85,B 0,C 180,E1 13826.752,E2 13826.752} C_VEL
LIN {X 0,Y 315.433,Z 614.557,A -85,B 0,C 180,E1 13826.308,E2 13826.308} C_VEL
LIN {X 0,Y 312.33,Z 627.823,A -85,B 0,C 180,E1 13823.766,E2 13823.766} C_VEL
LIN {X 0,Y 313.413,Z 634.203,A -85,B 0,C 180,E1 13823.275,E2 13823.275} C_VEL
LIN {X 0,Y 318.874,Z 663.314,A -85,B 0,C 180,E1 13821.435,E2 13821.435} C_VEL
LIN {X 0,Y 320.598,Z 675.891,A -85,B 0,C 180,E1 13820.774,E2 13820.774} C_VEL
LIN {X 0,Y 316.435,Z 763.635,A -85,B 0,C 180,E1 13818.611,E2 13818.611} C_VEL
LIN {X 0,Y 315.217,Z 779.71,A -85,B 0,C 180,E1 13817.897,E2 13817.897} C_VEL
LIN {X 0,Y 313.468,Z 794.755,A -85,B 0,C 180,E1 13816.914,E2 13816.914} C_VEL
LIN {X 0,Y 311.102,Z 809.517,A -85,B 0,C 180,E1 13815.594,E2 13815.594} C_VEL
LIN {X 0,Y 308.296,Z 823.594,A -85,B 0,C 180,E1 13813.943,E2 13813.943} C_VEL
LIN {X 0,Y 305.297,Z 836.079,A -85,B 0,C 180,E1 13812.04,E2 13812.04} C_VEL
LIN {X 0,Y 302.329,Z 847.18,A -85,B 0,C 180,E1 13809.89,E2 13809.89} C_VEL
LIN {X 0,Y 299.359,Z 857.037,A -85,B 0,C 180,E1 13807.43,E2 13807.43} C_VEL
LIN {X 0,Y 296.655,Z 865.42,A -85,B 0,C 180,E1 13804.716,E2 13804.716} C_VEL
LIN {X 0,Y 294.328,Z 872.108,A -85,B 0,C 180,E1 13801.767,E2 13801.767} C_VEL
LIN {X 0,Y 292.619,Z 876.854,A -85,B 0,C 180,E1 13798.797,E2 13798.797} C_VEL
LIN {X 0,Y 291.34,Z 879.996,A -85,B 0,C 180,E1 13795.497,E2 13795.497} C_VEL
LIN {X 0,Y 290.664,Z 881.183,A -85,B 0,C 180,E1 13792.442,E2 13792.442} C_VEL
LIN {X 0,Y 290.39,Z 880.575,A -85,B 0,C 180,E1 13789.089,E2 13789.089} C_VEL
LIN {X 0,Y 290.553,Z 878.284,A -85,B 0,C 180,E1 13785.976,E2 13785.976} C_VEL
LIN {X 0,Y 291.178,Z 873.88,A -85,B 0,C 180,E1 13782.692,E2 13782.692} C_VEL
LIN {X 0,Y 292.189,Z 868.033,A -85,B 0,C 180,E1 13779.758,E2 13779.758} C_VEL
LIN {X 0,Y 293.697,Z 860.135,A -85,B 0,C 180,E1 13776.84,E2 13776.84} C_VEL
LIN {X 0,Y 295.479,Z 850.947,A -85,B 0,C 180,E1 13774.267,E2 13774.267} C_VEL
LIN {X 0,Y 297.491,Z 840.341,A -85,B 0,C 180,E1 13771.924,E2 13771.924} C_VEL
LIN {X 0,Y 299.614,Z 828.09,A -85,B 0,C 180,E1 13769.806,E2 13769.806} C_VEL
LIN {X 0,Y 301.695,Z 814.834,A -85,B 0,C 180,E1 13768.004,E2 13768.004} C_VEL
LIN {X 0,Y 303.696,Z 799.475,A -85,B 0,C 180,E1 13766.412,E2 13766.412} C_VEL
LIN {X 0,Y 305.212,Z 784.364,A -85,B 0,C 180,E1 13765.253,E2 13765.253} C_VEL
LIN {X 0,Y 306.358,Z 767.931,A -85,B 0,C 180,E1 13764.373,E2 13764.373} C_VEL
LIN {X 0,Y 307.055,Z 748.353,A -85,B 0,C 180,E1 13763.768,E2 13763.768} C_VEL
LIN {X 0,Y 309.654,Z 669.995,A -85,B 0,C 180,E1 13761.883,E2 13761.883} C_VEL
LIN {X 0,Y 303.317,Z 628.247,A -85,B 0,C 180,E1 13760.033,E2 13760.033} C_VEL
LIN {X 0,Y 307.895,Z 601.778,A -85,B 0,C 180,E1 13755.134,E2 13755.134} C_VEL
LIN {X 0,Y 305.958,Z 592.408,A -85,B 0,C 180,E1 13752.895,E2 13752.895} C_VEL
LIN {X 0,Y 302.069,Z 577.551,A -85,B 0,C 180,E1 13749.054,E2 13749.054} C_VEL
LIN {X 0,Y 297.885,Z 563.887,A -85,B 0,C 180,E1 13745.193,E2 13745.193} C_VEL
LIN {X 0,Y 293.666,Z 551.91,A -85,B 0,C 180,E1 13741.454,E2 13741.454} C_VEL
LIN {X 0,Y 290.305,Z 542.747,A -85,B 0,C 180,E1 13738.252,E2 13738.252} C_VEL
LIN {X 0,Y 290.305,Z 542.579,A -85,B 0,C 180,E1 13737.065,E2 13737.065} C_VEL
LIN {X 0,Y 289.492,Z 542.73,A -85,B 0,C 180,E1 13735.652,E2 13735.652} C_VEL
LIN {X 0,Y 285.862,Z 543.193,A -85,B 0,C 180,E1 13733.311,E2 13733.311} C_VEL
LIN {X 0,Y 282.652,Z 543.594,A -85,B 0,C 180,E1 13730.897,E2 13730.897} C_VEL
LIN {X 0,Y 282.356,Z 543.628,A -85,B 0,C 180,E1 13730.101,E2 13730.101} C_VEL
LIN {X 0,Y 282.353,Z 543.614,A -85,B 0,C 180,E1 13725.38,E2 13725.38} C_VEL
LIN {X 0,Y 282.372,Z 543.585,A -85,B 0,C 180,E1 13720.658,E2 13720.658} C_VEL
LIN {X 0,Y 282.38,Z 543.602,A -85,B 0,C 180,E1 13716.169,E2 13716.169} C_VEL
LIN {X 0,Y 282.362,Z 543.612,A -85,B 0,C 180,E1 13711.421,E2 13711.421} C_VEL
LIN {X 0,Y 282.359,Z 543.576,A -85,B 0,C 180,E1 13706.726,E2 13706.726} C_VEL
LIN {X 0,Y 282.393,Z 543.622,A -85,B 0,C 180,E1 13702.044,E2 13702.044} C_VEL
LIN {X 0,Y 282.375,Z 543.568,A -85,B 0,C 180,E1 13697.304,E2 13697.304} C_VEL
LIN {X 0,Y 282.368,Z 543.623,A -85,B 0,C 180,E1 13692.682,E2 13692.682} C_VEL
LIN {X 0,Y 282.372,Z 543.57,A -85,B 0,C 180,E1 13687.938,E2 13687.938} C_VEL
LIN {X 0,Y 282.393,Z 543.608,A -85,B 0,C 180,E1 13683.248,E2 13683.248} C_VEL
LIN {X 0,Y 282.378,Z 543.585,A -85,B 0,C 180,E1 13678.58,E2 13678.58} C_VEL
LIN {X 0,Y 282.37,Z 543.59,A -85,B 0,C 180,E1 13673.902,E2 13673.902} C_VEL
LIN {X 0,Y 282.395,Z 543.619,A -85,B 0,C 180,E1 13669.184,E2 13669.184} C_VEL
LIN {X 0,Y 282.408,Z 543.582,A -85,B 0,C 180,E1 13664.602,E2 13664.602} C_VEL
LIN {X 0,Y 282.385,Z 543.595,A -85,B 0,C 180,E1 13659.913,E2 13659.913} C_VEL
LIN {X 0,Y 282.387,Z 543.609,A -85,B 0,C 180,E1 13655.081,E2 13655.081} C_VEL
LIN {X 0,Y 282.41,Z 543.615,A -85,B 0,C 180,E1 13650.52,E2 13650.52} C_VEL
LIN {X 0,Y 282.442,Z 543.935,A -85,B 0,C 180,E1 13648.805,E2 13648.805} C_VEL
LIN {X 0,Y 287.418,Z 555.81,A -85,B 0,C 180,E1 13644.971,E2 13644.971} C_VEL
LIN {X 0,Y 292.559,Z 568.807,A -85,B 0,C 180,E1 13641.287,E2 13641.287} C_VEL
LIN {X 0,Y 297.887,Z 583.683,A -85,B 0,C 180,E1 13637.573,E2 13637.573} C_VEL
LIN {X 0,Y 303.362,Z 600.672,A -85,B 0,C 180,E1 13633.796,E2 13633.796} C_VEL
LIN {X 0,Y 306.465,Z 611.485,A -85,B 0,C 180,E1 13631.611,E2 13631.611} C_VEL
LIN {X 0,Y 304.939,Z 619.532,A -85,B 0,C 180,E1 13630.559,E2 13630.559} C_VEL
LIN {X 0,Y 307.701,Z 655.312,A -85,B 0,C 180,E1 13629.292,E2 13629.292} C_VEL
LIN {X 0,Y 302.568,Z 806.085,A -85,B 0,C 180,E1 13625.862,E2 13625.862} C_VEL
LIN {X 0,Y 301.111,Z 824.394,A -85,B 0,C 180,E1 13625.125,E2 13625.125} C_VEL
LIN {X 0,Y 298.979,Z 842.277,A -85,B 0,C 180,E1 13624.066,E2 13624.066} C_VEL
LIN {X 0,Y 296.41,Z 859.616,A -85,B 0,C 180,E1 13622.664,E2 13622.664} C_VEL
LIN {X 0,Y 293.655,Z 875.975,A -85,B 0,C 180,E1 13620.94,E2 13620.94} C_VEL
LIN {X 0,Y 290.797,Z 891.326,A -85,B 0,C 180,E1 13618.887,E2 13618.887} C_VEL
LIN {X 0,Y 288.002,Z 905.697,A -85,B 0,C 180,E1 13616.495,E2 13616.495} C_VEL
LIN {X 0,Y 285.5,Z 919.035,A -85,B 0,C 180,E1 13613.75,E2 13613.75} C_VEL
LIN {X 0,Y 283.495,Z 930.567,A -85,B 0,C 180,E1 13610.832,E2 13610.832} C_VEL
LIN {X 0,Y 282.008,Z 941.087,A -85,B 0,C 180,E1 13607.541,E2 13607.541} C_VEL
LIN {X 0,Y 281.24,Z 949.552,A -85,B 0,C 180,E1 13604.201,E2 13604.201} C_VEL
LIN {X 0,Y 281.099,Z 956.47,A -85,B 0,C 180,E1 13600.661,E2 13600.661} C_VEL
LIN {X 0,Y 281.437,Z 961.477,A -85,B 0,C 180,E1 13597.145,E2 13597.145} C_VEL
LIN {X 0,Y 281.926,Z 964.553,A -85,B 0,C 180,E1 13593.866,E2 13593.866} C_VEL
LIN {X 0,Y 282.193,Z 965.971,A -85,B 0,C 180,E1 13590.814,E2 13590.814} C_VEL
LIN {X 0,Y 282.034,Z 966.003,A -85,B 0,C 180,E1 13587.768,E2 13587.768} C_VEL
LIN {X 0,Y 281.514,Z 964.574,A -85,B 0,C 180,E1 13584.5,E2 13584.5} C_VEL
LIN {X 0,Y 280.977,Z 961.198,A -85,B 0,C 180,E1 13580.789,E2 13580.789} C_VEL
LIN {X 0,Y 280.902,Z 955.955,A -85,B 0,C 180,E1 13577.045,E2 13577.045} C_VEL
LIN {X 0,Y 281.563,Z 949.199,A -85,B 0,C 180,E1 13573.495,E2 13573.495} C_VEL
LIN {X 0,Y 283.064,Z 940.56,A -85,B 0,C 180,E1 13569.967,E2 13569.967} C_VEL
LIN {X 0,Y 285.452,Z 930.107,A -85,B 0,C 180,E1 13566.593,E2 13566.593} C_VEL
LIN {X 0,Y 288.347,Z 918.771,A -85,B 0,C 180,E1 13563.656,E2 13563.656} C_VEL
LIN {X 0,Y 291.837,Z 905.6,A -85,B 0,C 180,E1 13560.895,E2 13560.895} C_VEL
LIN {X 0,Y 295.797,Z 890.832,A -85,B 0,C 180,E1 13558.409,E2 13558.409} C_VEL
LIN {X 0,Y 299.586,Z 875.606,A -85,B 0,C 180,E1 13556.363,E2 13556.363} C_VEL
LIN {X 0,Y 303.195,Z 859.702,A -85,B 0,C 180,E1 13554.68,E2 13554.68} C_VEL
LIN {X 0,Y 306.423,Z 843.281,A -85,B 0,C 180,E1 13553.342,E2 13553.342} C_VEL
LIN {X 0,Y 309.245,Z 825.497,A -85,B 0,C 180,E1 13552.281,E2 13552.281} C_VEL
LIN {X 0,Y 311.239,Z 807.425,A -85,B 0,C 180,E1 13551.536,E2 13551.536} C_VEL
LIN {X 0,Y 312.548,Z 782.264,A -85,B 0,C 180,E1 13550.9,E2 13550.9} C_VEL
LIN {X 0,Y 318.031,Z 653.917,A -85,B 0,C 180,E1 13547.962,E2 13547.962} C_VEL
LIN {X 0,Y 315.427,Z 624.745,A -85,B 0,C 180,E1 13546.609,E2 13546.609} C_VEL
LIN {X 0,Y 314.841,Z 621.198,A -85,B 0,C 180,E1 13546.391,E2 13546.391} C_VEL
LIN {X 0,Y 313.904,Z 618.679,A -85,B 0,C 180,E1 13545.912,E2 13545.912} C_VEL
LIN {X 0,Y 310.323,Z 606.542,A -85,B 0,C 180,E1 13542.734,E2 13542.734} C_VEL
LIN {X 0,Y 306.387,Z 595.302,A -85,B 0,C 180,E1 13539.279,E2 13539.279} C_VEL
LIN {X 0,Y 302.604,Z 585.666,A -85,B 0,C 180,E1 13535.791,E2 13535.791} C_VEL
LIN {X 0,Y 299.325,Z 578.054,A -85,B 0,C 180,E1 13532.534,E2 13532.534} C_VEL
LIN {X 0,Y 296.662,Z 571.863,A -85,B 0,C 180,E1 13529.477,E2 13529.477} C_VEL
LIN {X 0,Y 294.336,Z 567.188,A -85,B 0,C 180,E1 13526.641,E2 13526.641} C_VEL
LIN {X 0,Y 292.275,Z 562.845,A -85,B 0,C 180,E1 13523.553,E2 13523.553} C_VEL
LIN {X 0,Y 290.122,Z 558.423,A -85,B 0,C 180,E1 13519.529,E2 13519.529} C_VEL
LIN {X 0,Y 287.874,Z 553.953,A -85,B 0,C 180,E1 13512.843,E2 13512.843} C_VEL
LIN {X 0,Y 287.102,Z 553.053,A -85,B 0,C 180,E1 13507.604,E2 13507.604} C_VEL
LIN {X 0,Y 287.617,Z 553.679,A -85,B 0,C 180,E1 13502.59,E2 13502.59} C_VEL
LIN {X 0,Y 288.254,Z 555.73,A -85,B 0,C 180,E1 13498.807,E2 13498.807} C_VEL
LIN {X 0,Y 289.979,Z 558.641,A -85,B 0,C 180,E1 13494.658,E2 13494.658} C_VEL
LIN {X 0,Y 291.974,Z 563.225,A -85,B 0,C 180,E1 13490.443,E2 13490.443} C_VEL
LIN {X 0,Y 293.846,Z 567.682,A -85,B 0,C 180,E1 13487.222,E2 13487.222} C_VEL
LIN {X 0,Y 295.502,Z 571.735,A -85,B 0,C 180,E1 13484.697,E2 13484.697} C_VEL
LIN {X 0,Y 297.938,Z 577.744,A -85,B 0,C 180,E1 13481.408,E2 13481.408} C_VEL
LIN {X 0,Y 301.083,Z 586.667,A -85,B 0,C 180,E1 13477.342,E2 13477.342} C_VEL
LIN {X 0,Y 303.997,Z 596.197,A -85,B 0,C 180,E1 13473.639,E2 13473.639} C_VEL
LIN {X 0,Y 306.754,Z 606.664,A -85,B 0,C 180,E1 13470.085,E2 13470.085} C_VEL
LIN {X 0,Y 308.786,Z 617.055,A -85,B 0,C 180,E1 13466.986,E2 13466.986} C_VEL
LIN {X 0,Y 306.164,Z 627.66,A -85,B 0,C 180,E1 13464.916,E2 13464.916} C_VEL
LIN {X 0,Y 308.11,Z 638.431,A -85,B 0,C 180,E1 13464.101,E2 13464.101} C_VEL
LIN {X 0,Y 313.231,Z 666.892,A -85,B 0,C 180,E1 13462.259,E2 13462.259} C_VEL
LIN {X 0,Y 314.535,Z 677.324,A -85,B 0,C 180,E1 13461.7,E2 13461.7} C_VEL
LIN {X 0,Y 310.202,Z 764.521,A -85,B 0,C 180,E1 13459.515,E2 13459.515} C_VEL
LIN {X 0,Y 308.897,Z 780.742,A -85,B 0,C 180,E1 13458.778,E2 13458.778} C_VEL
LIN {X 0,Y 307.073,Z 795.637,A -85,B 0,C 180,E1 13457.787,E2 13457.787} C_VEL
LIN {X 0,Y 304.661,Z 810.027,A -85,B 0,C 180,E1 13456.485,E2 13456.485} C_VEL
LIN {X 0,Y 301.663,Z 824.393,A -85,B 0,C 180,E1 13454.78,E2 13454.78} C_VEL
LIN {X 0,Y 298.491,Z 836.972,A -85,B 0,C 180,E1 13452.835,E2 13452.835} C_VEL
LIN {X 0,Y 295.229,Z 848.513,A -85,B 0,C 180,E1 13450.553,E2 13450.553} C_VEL
LIN {X 0,Y 292.084,Z 858.354,A -85,B 0,C 180,E1 13448.03,E2 13448.03} C_VEL
LIN {X 0,Y 289.222,Z 866.684,A -85,B 0,C 180,E1 13445.256,E2 13445.256} C_VEL
LIN {X 0,Y 286.745,Z 873.335,A -85,B 0,C 180,E1 13442.236,E2 13442.236} C_VEL
LIN {X 0,Y 284.911,Z 878.054,A -85,B 0,C 180,E1 13439.191,E2 13439.191} C_VEL
LIN {X 0,Y 283.565,Z 881.105,A -85,B 0,C 180,E1 13435.922,E2 13435.922} C_VEL
LIN {X 0,Y 282.787,Z 882.38,A -85,B 0,C 180,E1 13432.656,E2 13432.656} C_VEL
LIN {X 0,Y 282.474,Z 881.779,A -85,B 0,C 180,E1 13429.215,E2 13429.215} C_VEL
LIN {X 0,Y 282.626,Z 879.515,A -85,B 0,C 180,E1 13426.014,E2 13426.014} C_VEL
LIN {X 0,Y 283.264,Z 875.13,A -85,B 0,C 180,E1 13422.638,E2 13422.638} C_VEL
LIN {X 0,Y 284.269,Z 869.553,A -85,B 0,C 180,E1 13419.716,E2 13419.716} C_VEL
LIN {X 0,Y 285.869,Z 861.466,A -85,B 0,C 180,E1 13416.621,E2 13416.621} C_VEL
LIN {X 0,Y 287.713,Z 852.377,A -85,B 0,C 180,E1 13413.983,E2 13413.983} C_VEL
LIN {X 0,Y 289.891,Z 841.374,A -85,B 0,C 180,E1 13411.48,E2 13411.48} C_VEL
LIN {X 0,Y 292.104,Z 829.138,A -85,B 0,C 180,E1 13409.311,E2 13409.311} C_VEL
LIN {X 0,Y 294.27,Z 815.928,A -85,B 0,C 180,E1 13407.466,E2 13407.466} C_VEL
LIN {X 0,Y 296.224,Z 801.64,A -85,B 0,C 180,E1 13405.933,E2 13405.933} C_VEL
LIN {X 0,Y 297.874,Z 786.414,A -85,B 0,C 180,E1 13404.702,E2 13404.702} C_VEL
LIN {X 0,Y 299.145,Z 769.272,A -85,B 0,C 180,E1 13403.744,E2 13403.744} C_VEL
LIN {X 0,Y 299.84,Z 751.404,A -85,B 0,C 180,E1 13403.155,E2 13403.155} C_VEL
LIN {X 0,Y 302.612,Z 670.958,A -85,B 0,C 180,E1 13401.176,E2 13401.176} C_VEL
LIN {X 0,Y 296.191,Z 628.35,A -85,B 0,C 180,E1 13399.249,E2 13399.249} C_VEL
LIN {X 0,Y 300.611,Z 603.673,A -85,B 0,C 180,E1 13394.617,E2 13394.617} C_VEL
LIN {X 0,Y 297.087,Z 588.77,A -85,B 0,C 180,E1 13390.843,E2 13390.843} C_VEL
LIN {X 0,Y 293.227,Z 574.885,A -85,B 0,C 180,E1 13387.024,E2 13387.024} C_VEL
LIN {X 0,Y 289.291,Z 562.57,A -85,B 0,C 180,E1 13383.3,E2 13383.3} C_VEL
LIN {X 0,Y 284.955,Z 550.471,A -85,B 0,C 180,E1 13379.28,E2 13379.28} C_VEL
LIN {X 0,Y 282.386,Z 543.744,A -85,B 0,C 180,E1 13376.714,E2 13376.714} C_VEL
LIN {X 0,Y 282.347,Z 543.604,A -85,B 0,C 180,E1 13371.963,E2 13371.963} C_VEL
LIN {X 0,Y 282.356,Z 543.628,A -85,B 0,C 180,E1 13370.101,E2 13370.101} C_VEL
LIN {X 0,Y 281.323,Z 543.754,A -85,B 0,C 180,E1 13368.538,E2 13368.538} C_VEL
LIN {X 0,Y 276.879,Z 544.312,A -85,B 0,C 180,E1 13365.688,E2 13365.688} C_VEL
LIN {X 0,Y 274.596,Z 544.586,A -85,B 0,C 180,E1 13363.639,E2 13363.639} C_VEL
LIN {X 0,Y 274.424,Z 544.591,A -85,B 0,C 180,E1 13362.938,E2 13362.938} C_VEL
LIN {X 0,Y 274.451,Z 544.607,A -85,B 0,C 180,E1 13358.268,E2 13358.268} C_VEL
LIN {X 0,Y 274.417,Z 544.569,A -85,B 0,C 180,E1 13353.452,E2 13353.452} C_VEL
LIN {X 0,Y 274.428,Z 544.594,A -85,B 0,C 180,E1 13348.594,E2 13348.594} C_VEL
LIN {X 0,Y 274.45,Z 544.583,A -85,B 0,C 180,E1 13343.853,E2 13343.853} C_VEL
LIN {X 0,Y 274.436,Z 544.572,A -85,B 0,C 180,E1 13339.338,E2 13339.338} C_VEL
LIN {X 0,Y 274.424,Z 544.599,A -85,B 0,C 180,E1 13334.561,E2 13334.561} C_VEL
LIN {X 0,Y 274.438,Z 544.559,A -85,B 0,C 180,E1 13329.86,E2 13329.86} C_VEL
LIN {X 0,Y 274.456,Z 544.603,A -85,B 0,C 180,E1 13325.226,E2 13325.226} C_VEL
LIN {X 0,Y 274.427,Z 544.557,A -85,B 0,C 180,E1 13320.418,E2 13320.418} C_VEL
LIN {X 0,Y 274.443,Z 544.609,A -85,B 0,C 180,E1 13315.613,E2 13315.613} C_VEL
LIN {X 0,Y 274.459,Z 544.572,A -85,B 0,C 180,E1 13310.988,E2 13310.988} C_VEL
LIN {X 0,Y 274.449,Z 544.577,A -85,B 0,C 180,E1 13306.302,E2 13306.302} C_VEL
LIN {X 0,Y 274.445,Z 544.611,A -85,B 0,C 180,E1 13301.521,E2 13301.521} C_VEL
LIN {X 0,Y 274.457,Z 544.597,A -85,B 0,C 180,E1 13296.831,E2 13296.831} C_VEL
LIN {X 0,Y 274.477,Z 544.586,A -85,B 0,C 180,E1 13292.208,E2 13292.208} C_VEL
LIN {X 0,Y 274.525,Z 544.965,A -85,B 0,C 180,E1 13290.51,E2 13290.51} C_VEL
LIN {X 0,Y 279.48,Z 556.62,A -85,B 0,C 180,E1 13286.465,E2 13286.465} C_VEL
LIN {X 0,Y 284.755,Z 569.768,A -85,B 0,C 180,E1 13282.516,E2 13282.516} C_VEL
LIN {X 0,Y 290.158,Z 584.753,A -85,B 0,C 180,E1 13278.577,E2 13278.577} C_VEL
LIN {X 0,Y 295.491,Z 601.411,A -85,B 0,C 180,E1 13274.718,E2 13274.718} C_VEL
LIN {X 0,Y 299.055,Z 614.035,A -85,B 0,C 180,E1 13272.078,E2 13272.078} C_VEL
LIN {X 0,Y 297.995,Z 619.721,A -85,B 0,C 180,E1 13271.342,E2 13271.342} C_VEL
LIN {X 0,Y 300.722,Z 656.026,A -85,B 0,C 180,E1 13270.022,E2 13270.022} C_VEL
LIN {X 0,Y 295.424,Z 805.405,A -85,B 0,C 180,E1 13266.56,E2 13266.56} C_VEL
LIN {X 0,Y 293.929,Z 823.697,A -85,B 0,C 180,E1 13265.809,E2 13265.809} C_VEL
LIN {X 0,Y 291.738,Z 841.498,A -85,B 0,C 180,E1 13264.734,E2 13264.734} C_VEL
LIN {X 0,Y 289.16,Z 858.304,A -85,B 0,C 180,E1 13263.352,E2 13263.352} C_VEL
LIN {X 0,Y 286.292,Z 874.75,A -85,B 0,C 180,E1 13261.592,E2 13261.592} C_VEL
LIN {X 0,Y 283.322,Z 890.178,A -85,B 0,C 180,E1 13259.492,E2 13259.492} C_VEL
LIN {X 0,Y 280.402,Z 904.576,A -85,B 0,C 180,E1 13257.042,E2 13257.042} C_VEL
LIN {X 0,Y 277.781,Z 917.932,A -85,B 0,C 180,E1 13254.227,E2 13254.227} C_VEL
LIN {X 0,Y 275.678,Z 929.456,A -85,B 0,C 180,E1 13251.234,E2 13251.234} C_VEL
LIN {X 0,Y 274.105,Z 939.994,A -85,B 0,C 180,E1 13247.844,E2 13247.844} C_VEL
LIN {X 0,Y 273.292,Z 948.469,A -85,B 0,C 180,E1 13244.407,E2 13244.407} C_VEL
LIN {X 0,Y 273.138,Z 955.381,A -85,B 0,C 180,E1 13240.761,E2 13240.761} C_VEL
LIN {X 0,Y 273.468,Z 960.146,A -85,B 0,C 180,E1 13237.354,E2 13237.354} C_VEL
LIN {X 0,Y 273.989,Z 963.288,A -85,B 0,C 180,E1 13233.978,E2 13233.978} C_VEL
LIN {X 0,Y 274.284,Z 964.745,A -85,B 0,C 180,E1 13230.838,E2 13230.838} C_VEL
LIN {X 0,Y 274.107,Z 964.821,A -85,B 0,C 180,E1 13227.703,E2 13227.703} C_VEL
LIN {X 0,Y 273.54,Z 963.428,A -85,B 0,C 180,E1 13224.339,E2 13224.339} C_VEL
LIN {X 0,Y 273.005,Z 960.329,A -85,B 0,C 180,E1 13220.73,E2 13220.73} C_VEL
LIN {X 0,Y 272.929,Z 955.223,A -85,B 0,C 180,E1 13216.875,E2 13216.875} C_VEL
LIN {X 0,Y 273.7,Z 948.171,A -85,B 0,C 180,E1 13213.012,E2 13213.012} C_VEL
LIN {X 0,Y 275.348,Z 939.557,A -85,B 0,C 180,E1 13209.381,E2 13209.381} C_VEL
LIN {X 0,Y 277.841,Z 929.461,A -85,B 0,C 180,E1 13206.01,E2 13206.01} C_VEL
LIN {X 0,Y 281.012,Z 917.883,A -85,B 0,C 180,E1 13202.913,E2 13202.913} C_VEL
LIN {X 0,Y 284.717,Z 904.798,A -85,B 0,C 180,E1 13200.094,E2 13200.094} C_VEL
LIN {X 0,Y 288.88,Z 890.079,A -85,B 0,C 180,E1 13197.562,E2 13197.562} C_VEL
LIN {X 0,Y 292.86,Z 874.899,A -85,B 0,C 180,E1 13195.483,E2 13195.483} C_VEL
LIN {X 0,Y 296.608,Z 859.154,A -85,B 0,C 180,E1 13193.788,E2 13193.788} C_VEL
LIN {X 0,Y 299.994,Z 842.698,A -85,B 0,C 180,E1 13192.423,E2 13192.423} C_VEL
LIN {X 0,Y 302.946,Z 824.9,A -85,B 0,C 180,E1 13191.346,E2 13191.346} C_VEL
LIN {X 0,Y 305.024,Z 806.737,A -85,B 0,C 180,E1 13190.587,E2 13190.587} C_VEL
LIN {X 0,Y 306.403,Z 781.35,A -85,B 0,C 180,E1 13189.937,E2 13189.937} C_VEL
LIN {X 0,Y 312.112,Z 654.833,A -85,B 0,C 180,E1 13186.99,E2 13186.99} C_VEL
LIN {X 0,Y 309.613,Z 625.578,A -85,B 0,C 180,E1 13185.585,E2 13185.585} C_VEL
LIN {X 0,Y 306.696,Z 619.938,A -85,B 0,C 180,E1 13184.763,E2 13184.763} C_VEL
LIN {X 0,Y 303.144,Z 608.304,A -85,B 0,C 180,E1 13181.525,E2 13181.525} C_VEL
LIN {X 0,Y 299.495,Z 597.943,A -85,B 0,C 180,E1 13178.142,E2 13178.142} C_VEL
LIN {X 0,Y 295.926,Z 588.698,A -85,B 0,C 180,E1 13174.585,E2 13174.585} C_VEL
LIN {X 0,Y 292.432,Z 580.672,A -85,B 0,C 180,E1 13170.855,E2 13170.855} C_VEL
LIN {X 0,Y 290.618,Z 576.709,A -85,B 0,C 180,E1 13168.694,E2 13168.694} C_VEL
LIN {X 0,Y 288.997,Z 573.108,A -85,B 0,C 180,E1 13166.507,E2 13166.507} C_VEL
LIN {X 0,Y 286.98,Z 568.805,A -85,B 0,C 180,E1 13163.402,E2 13163.402} C_VEL
LIN {X 0,Y 284.818,Z 564.368,A -85,B 0,C 180,E1 13159.268,E2 13159.268} C_VEL
LIN {X 0,Y 282.715,Z 560.053,A -85,B 0,C 180,E1 13152.666,E2 13152.666} C_VEL
LIN {X 0,Y 281.97,Z 559.178,A -85,B 0,C 180,E1 13147.334,E2 13147.334} C_VEL
LIN {X 0,Y 282.506,Z 559.879,A -85,B 0,C 180,E1 13142.231,E2 13142.231} C_VEL
LIN {X 0,Y 284.53,Z 564.318,A -85,B 0,C 180,E1 13134.96,E2 13134.96} C_VEL
LIN {X 0,Y 286.464,Z 569.034,A -85,B 0,C 180,E1 13130.558,E2 13130.558} C_VEL
LIN {X 0,Y 288.103,Z 572.978,A -85,B 0,C 180,E1 13127.574,E2 13127.574} C_VEL
LIN {X 0,Y 289.932,Z 577.718,A -85,B 0,C 180,E1 13124.6,E2 13124.6} C_VEL
LIN {X 0,Y 292.137,Z 583.453,A -85,B 0,C 180,E1 13121.429,E2 13121.429} C_VEL
LIN {X 0,Y 295.208,Z 592.406,A -85,B 0,C 180,E1 13117.287,E2 13117.287} C_VEL
LIN {X 0,Y 298.03,Z 602.013,A -85,B 0,C 180,E1 13113.499,E2 13113.499} C_VEL
LIN {X 0,Y 300.61,Z 612.739,A -85,B 0,C 180,E1 13109.851,E2 13109.851} C_VEL
LIN {X 0,Y 302.023,Z 620.219,A -85,B 0,C 180,E1 13107.567,E2 13107.567} C_VEL
LIN {X 0,Y 300.108,Z 627.876,A -85,B 0,C 180,E1 13106.078,E2 13106.078} C_VEL
LIN {X 0,Y 305.466,Z 656.898,A -85,B 0,C 180,E1 13103.973,E2 13103.973} C_VEL
LIN {X 0,Y 308.637,Z 678.173,A -85,B 0,C 180,E1 13102.685,E2 13102.685} C_VEL
LIN {X 0,Y 304.106,Z 765.079,A -85,B 0,C 180,E1 13100.476,E2 13100.476} C_VEL
LIN {X 0,Y 302.739,Z 781.278,A -85,B 0,C 180,E1 13099.732,E2 13099.732} C_VEL
LIN {X 0,Y 300.761,Z 796.615,A -85,B 0,C 180,E1 13098.696,E2 13098.696} C_VEL
LIN {X 0,Y 298.218,Z 810.984,A -85,B 0,C 180,E1 13097.369,E2 13097.369} C_VEL
LIN {X 0,Y 295.062,Z 825.344,A -85,B 0,C 180,E1 13095.635,E2 13095.635} C_VEL
LIN {X 0,Y 291.789,Z 837.711,A -85,B 0,C 180,E1 13093.695,E2 13093.695} C_VEL
LIN {X 0,Y 288.448,Z 848.952,A -85,B 0,C 180,E1 13091.45,E2 13091.45} C_VEL
LIN {X 0,Y 285.101,Z 858.939,A -85,B 0,C 180,E1 13088.878,E2 13088.878} C_VEL
LIN {X 0,Y 282.03,Z 867.39,A -85,B 0,C 180,E1 13086.044,E2 13086.044} C_VEL
LIN {X 0,Y 279.515,Z 873.762,A -85,B 0,C 180,E1 13083.17,E2 13083.17} C_VEL
LIN {X 0,Y 277.338,Z 878.989,A -85,B 0,C 180,E1 13079.83,E2 13079.83} C_VEL
LIN {X 0,Y 275.844,Z 882.163,A -85,B 0,C 180,E1 13076.472,E2 13076.472} C_VEL
LIN {X 0,Y 274.946,Z 883.551,A -85,B 0,C 180,E1 13073.065,E2 13073.065} C_VEL
LIN {X 0,Y 274.576,Z 883.161,A -85,B 0,C 180,E1 13069.791,E2 13069.791} C_VEL
LIN {X 0,Y 274.676,Z 880.936,A -85,B 0,C 180,E1 13066.273,E2 13066.273} C_VEL
LIN {X 0,Y 275.237,Z 877.027,A -85,B 0,C 180,E1 13063.013,E2 13063.013} C_VEL
LIN {X 0,Y 276.297,Z 871.299,A -85,B 0,C 180,E1 13059.789,E2 13059.789} C_VEL
LIN {X 0,Y 277.782,Z 864.008,A -85,B 0,C 180,E1 13056.819,E2 13056.819} C_VEL
LIN {X 0,Y 279.664,Z 855.184,A -85,B 0,C 180,E1 13054.056,E2 13054.056} C_VEL
LIN {X 0,Y 281.721,Z 845.25,A -85,B 0,C 180,E1 13051.624,E2 13051.624} C_VEL
LIN {X 0,Y 283.98,Z 833.673,A -85,B 0,C 180,E1 13049.374,E2 13049.374} C_VEL
LIN {X 0,Y 286.128,Z 821.477,A -85,B 0,C 180,E1 13047.494,E2 13047.494} C_VEL
LIN {X 0,Y 288.388,Z 806.671,A -85,B 0,C 180,E1 13045.723,E2 13045.723} C_VEL
LIN {X 0,Y 290.089,Z 792.781,A -85,B 0,C 180,E1 13044.46,E2 13044.46} C_VEL
LIN {X 0,Y 291.599,Z 775.973,A -85,B 0,C 180,E1 13043.353,E2 13043.353} C_VEL
LIN {X 0,Y 292.479,Z 759.447,A -85,B 0,C 180,E1 13042.664,E2 13042.664} C_VEL
LIN {X 0,Y 295.596,Z 671.955,A -85,B 0,C 180,E1 13040.446,E2 13040.446} C_VEL
LIN {X 0,Y 289.105,Z 627.926,A -85,B 0,C 180,E1 13038.376,E2 13038.376} C_VEL
LIN {X 0,Y 293.234,Z 606.094,A -85,B 0,C 180,E1 13034.169,E2 13034.169} C_VEL
LIN {X 0,Y 289.816,Z 591.445,A -85,B 0,C 180,E1 13030.366,E2 13030.366} C_VEL
LIN {X 0,Y 286.051,Z 577.853,A -85,B 0,C 180,E1 13026.517,E2 13026.517} C_VEL
LIN {X 0,Y 282.224,Z 565.881,A -85,B 0,C 180,E1 13022.779,E2 13022.779} C_VEL
LIN {X 0,Y 278.273,Z 554.679,A -85,B 0,C 180,E1 13018.95,E2 13018.95} C_VEL
LIN {X 0,Y 275.252,Z 547.294,A -85,B 0,C 180,E1 13016.103,E2 13016.103} C_VEL
LIN {X 0,Y 274.442,Z 544.677,A -85,B 0,C 180,E1 13014.997,E2 13014.997} C_VEL
LIN {X 0,Y 274.423,Z 544.617,A -85,B 0,C 180,E1 13010.245,E2 13010.245} C_VEL
LIN {X 0,Y 274.412,Z 544.598,A -85,B 0,C 180,E1 13005.575,E2 13005.575} C_VEL
LIN {X 0,Y 274.424,Z 544.591,A -85,B 0,C 180,E1 13002.938,E2 13002.938} C_VEL
LIN {X 0,Y 273.612,Z 544.679,A -85,B 0,C 180,E1 13001.442,E2 13001.442} C_VEL
LIN {X 0,Y 270.166,Z 545.125,A -85,B 0,C 180,E1 12999.077,E2 12999.077} C_VEL
LIN {X 0,Y 266.855,Z 545.543,A -85,B 0,C 180,E1 12996.524,E2 12996.524} C_VEL
LIN {X 0,Y 266.48,Z 545.568,A -85,B 0,C 180,E1 12995.561,E2 12995.561} C_VEL
LIN {X 0,Y 266.49,Z 545.6,A -85,B 0,C 180,E1 12990.682,E2 12990.682} C_VEL
LIN {X 0,Y 266.503,Z 545.546,A -85,B 0,C 180,E1 12986.038,E2 12986.038} C_VEL
LIN {X 0,Y 266.499,Z 545.599,A -85,B 0,C 180,E1 12981.342,E2 12981.342} C_VEL
LIN {X 0,Y 266.485,Z 545.552,A -85,B 0,C 180,E1 12976.344,E2 12976.344} C_VEL
LIN {X 0,Y 266.509,Z 545.581,A -85,B 0,C 180,E1 12971.689,E2 12971.689} C_VEL
LIN {X 0,Y 266.498,Z 545.559,A -85,B 0,C 180,E1 12966.896,E2 12966.896} C_VEL
LIN {X 0,Y 266.489,Z 545.561,A -85,B 0,C 180,E1 12962.151,E2 12962.151} C_VEL
LIN {X 0,Y 266.509,Z 545.586,A -85,B 0,C 180,E1 12957.42,E2 12957.42} C_VEL
LIN {X 0,Y 266.516,Z 545.55,A -85,B 0,C 180,E1 12952.672,E2 12952.672} C_VEL
LIN {X 0,Y 266.501,Z 545.594,A -85,B 0,C 180,E1 12947.872,E2 12947.872} C_VEL
LIN {X 0,Y 266.517,Z 545.582,A -85,B 0,C 180,E1 12942.985,E2 12942.985} C_VEL
LIN {X 0,Y 266.522,Z 545.566,A -85,B 0,C 180,E1 12938.198,E2 12938.198} C_VEL
LIN {X 0,Y 266.507,Z 545.571,A -85,B 0,C 180,E1 12933.484,E2 12933.484} C_VEL
LIN {X 0,Y 266.597,Z 545.976,A -85,B 0,C 180,E1 12932.372,E2 12932.372} C_VEL
LIN {X 0,Y 268.229,Z 549.67,A -85,B 0,C 180,E1 12930.892,E2 12930.892} C_VEL
LIN {X 0,Y 273.241,Z 561.543,A -85,B 0,C 180,E1 12926.71,E2 12926.71} C_VEL
LIN {X 0,Y 278.207,Z 574.049,A -85,B 0,C 180,E1 12922.859,E2 12922.859} C_VEL
LIN {X 0,Y 283.601,Z 589.31,A -85,B 0,C 180,E1 12918.755,E2 12918.755} C_VEL
LIN {X 0,Y 288.867,Z 606.089,A -85,B 0,C 180,E1 12914.801,E2 12914.801} C_VEL
LIN {X 0,Y 291.714,Z 616.316,A -85,B 0,C 180,E1 12912.603,E2 12912.603} C_VEL
LIN {X 0,Y 291.091,Z 619.999,A -85,B 0,C 180,E1 12912.15,E2 12912.15} C_VEL
LIN {X 0,Y 293.763,Z 656.805,A -85,B 0,C 180,E1 12910.776,E2 12910.776} C_VEL
LIN {X 0,Y 288.289,Z 804.814,A -85,B 0,C 180,E1 12907.276,E2 12907.276} C_VEL
LIN {X 0,Y 286.749,Z 823.139,A -85,B 0,C 180,E1 12906.508,E2 12906.508} C_VEL
LIN {X 0,Y 284.425,Z 841.359,A -85,B 0,C 180,E1 12905.381,E2 12905.381} C_VEL
LIN {X 0,Y 281.781,Z 857.973,A -85,B 0,C 180,E1 12903.977,E2 12903.977} C_VEL
LIN {X 0,Y 278.846,Z 874.183,A -85,B 0,C 180,E1 12902.197,E2 12902.197} C_VEL
LIN {X 0,Y 275.741,Z 889.67,A -85,B 0,C 180,E1 12900.026,E2 12900.026} C_VEL
LIN {X 0,Y 272.712,Z 903.99,A -85,B 0,C 180,E1 12897.514,E2 12897.514} C_VEL
LIN {X 0,Y 270.08,Z 916.826,A -85,B 0,C 180,E1 12894.73,E2 12894.73} C_VEL
LIN {X 0,Y 267.875,Z 928.345,A -85,B 0,C 180,E1 12891.658,E2 12891.658} C_VEL
LIN {X 0,Y 266.292,Z 938.287,A -85,B 0,C 180,E1 12888.386,E2 12888.386} C_VEL
LIN {X 0,Y 265.383,Z 946.884,A -85,B 0,C 180,E1 12884.846,E2 12884.846} C_VEL
LIN {X 0,Y 265.167,Z 953.938,A -85,B 0,C 180,E1 12881.089,E2 12881.089} C_VEL
LIN {X 0,Y 265.531,Z 959.022,A -85,B 0,C 180,E1 12877.358,E2 12877.358} C_VEL
LIN {X 0,Y 266.084,Z 962.146,A -85,B 0,C 180,E1 12873.881,E2 12873.881} C_VEL
LIN {X 0,Y 266.381,Z 963.577,A -85,B 0,C 180,E1 12870.648,E2 12870.648} C_VEL
LIN {X 0,Y 266.148,Z 963.601,A -85,B 0,C 180,E1 12867.419,E2 12867.419} C_VEL
LIN {X 0,Y 265.522,Z 962.146,A -85,B 0,C 180,E1 12863.951,E2 12863.951} C_VEL
LIN {X 0,Y 264.973,Z 958.744,A -85,B 0,C 180,E1 12860.008,E2 12860.008} C_VEL
LIN {X 0,Y 265.027,Z 953.472,A -85,B 0,C 180,E1 12856.032,E2 12856.032} C_VEL
LIN {X 0,Y 265.932,Z 946.691,A -85,B 0,C 180,E1 12852.274,E2 12852.274} C_VEL
LIN {X 0,Y 267.801,Z 938.016,A -85,B 0,C 180,E1 12848.542,E2 12848.542} C_VEL
LIN {X 0,Y 270.544,Z 927.846,A -85,B 0,C 180,E1 12845.088,E2 12845.088} C_VEL
LIN {X 0,Y 273.975,Z 916.164,A -85,B 0,C 180,E1 12841.921,E2 12841.921} C_VEL
LIN {X 0,Y 277.973,Z 902.96,A -85,B 0,C 180,E1 12839.051,E2 12839.051} C_VEL
LIN {X 0,Y 282.213,Z 888.704,A -85,B 0,C 180,E1 12836.576,E2 12836.576} C_VEL
LIN {X 0,Y 286.412,Z 873.445,A -85,B 0,C 180,E1 12834.468,E2 12834.468} C_VEL
LIN {X 0,Y 290.44,Z 857.166,A -85,B 0,C 180,E1 12832.714,E2 12832.714} C_VEL
LIN {X 0,Y 293.885,Z 840.896,A -85,B 0,C 180,E1 12831.376,E2 12831.376} C_VEL
LIN {X 0,Y 296.889,Z 823.328,A -85,B 0,C 180,E1 12830.318,E2 12830.318} C_VEL
LIN {X 0,Y 299.02,Z 804.993,A -85,B 0,C 180,E1 12829.556,E2 12829.556} C_VEL
LIN {X 0,Y 300.52,Z 777.608,A -85,B 0,C 180,E1 12828.861,E2 12828.861} C_VEL
LIN {X 0,Y 306.306,Z 655.858,A -85,B 0,C 180,E1 12825.982,E2 12825.982} C_VEL
LIN {X 0,Y 304.148,Z 629.43,A -85,B 0,C 180,E1 12824.675,E2 12824.675} C_VEL
LIN {X 0,Y 299.351,Z 620.61,A -85,B 0,C 180,E1 12823.345,E2 12823.345} C_VEL
LIN {X 0,Y 295.966,Z 609.911,A -85,B 0,C 180,E1 12820.184,E2 12820.184} C_VEL
LIN {X 0,Y 292.476,Z 600.137,A -85,B 0,C 180,E1 12816.745,E2 12816.745} C_VEL
LIN {X 0,Y 288.917,Z 590.918,A -85,B 0,C 180,E1 12812.91,E2 12812.91} C_VEL
LIN {X 0,Y 285.731,Z 583.406,A -85,B 0,C 180,E1 12809.104,E2 12809.104} C_VEL
LIN {X 0,Y 283.478,Z 578.76,A -85,B 0,C 180,E1 12806.16,E2 12806.16} C_VEL
LIN {X 0,Y 281.657,Z 574.725,A -85,B 0,C 180,E1 12803.206,E2 12803.206} C_VEL
LIN {X 0,Y 279.64,Z 570.459,A -85,B 0,C 180,E1 12799.205,E2 12799.205} C_VEL
LIN {X 0,Y 277.572,Z 566.173,A -85,B 0,C 180,E1 12792.564,E2 12792.564} C_VEL
LIN {X 0,Y 276.831,Z 565.311,A -85,B 0,C 180,E1 12787.262,E2 12787.262} C_VEL
LIN {X 0,Y 277.342,Z 566.023,A -85,B 0,C 180,E1 12782.066,E2 12782.066} C_VEL
LIN {X 0,Y 279.202,Z 570.479,A -85,B 0,C 180,E1 12774.863,E2 12774.863} C_VEL
LIN {X 0,Y 280.921,Z 574.695,A -85,B 0,C 180,E1 12770.783,E2 12770.783} C_VEL
LIN {X 0,Y 282.568,Z 578.963,A -85,B 0,C 180,E1 12767.534,E2 12767.534} C_VEL
LIN {X 0,Y 284.376,Z 583.68,A -85,B 0,C 180,E1 12764.501,E2 12764.501} C_VEL
LIN {X 0,Y 286.779,Z 590.344,A -85,B 0,C 180,E1 12760.86,E2 12760.86} C_VEL
LIN {X 0,Y 289.469,Z 598.615,A -85,B 0,C 180,E1 12757.025,E2 12757.025} C_VEL
LIN {X 0,Y 292.16,Z 608.473,A -85,B 0,C 180,E1 12753.144,E2 12753.144} C_VEL
LIN {X 0,Y 294.481,Z 618.943,A -85,B 0,C 180,E1 12749.575,E2 12749.575} C_VEL
LIN {X 0,Y 295.199,Z 623.764,A -85,B 0,C 180,E1 12748.103,E2 12748.103} C_VEL
LIN {X 0,Y 294.26,Z 627.256,A -85,B 0,C 180,E1 12747.411,E2 12747.411} C_VEL
LIN {X 0,Y 295.175,Z 633.207,A -85,B 0,C 180,E1 12746.878,E2 12746.878} C_VEL
LIN {X 0,Y 300.337,Z 662.042,A -85,B 0,C 180,E1 12744.776,E2 12744.776} C_VEL
LIN {X 0,Y 302.791,Z 679.791,A -85,B 0,C 180,E1 12743.689,E2 12743.689} C_VEL
LIN {X 0,Y 298.105,Z 765.791,A -85,B 0,C 180,E1 12741.474,E2 12741.474} C_VEL
LIN {X 0,Y 296.679,Z 781.919,A -85,B 0,C 180,E1 12740.723,E2 12740.723} C_VEL
LIN {X 0,Y 294.519,Z 797.849,A -85,B 0,C 180,E1 12739.63,E2 12739.63} C_VEL
LIN {X 0,Y 291.684,Z 812.91,A -85,B 0,C 180,E1 12738.198,E2 12738.198} C_VEL
LIN {X 0,Y 288.564,Z 826.339,A -85,B 0,C 180,E1 12736.535,E2 12736.535} C_VEL
LIN {X 0,Y 285.074,Z 838.824,A -85,B 0,C 180,E1 12734.537,E2 12734.537} C_VEL
LIN {X 0,Y 281.437,Z 850.377,A -85,B 0,C 180,E1 12732.172,E2 12732.172} C_VEL
LIN {X 0,Y 277.91,Z 860.254,A -85,B 0,C 180,E1 12729.547,E2 12729.547} C_VEL
LIN {X 0,Y 274.668,Z 868.662,A -85,B 0,C 180,E1 12726.648,E2 12726.648} C_VEL
LIN {X 0,Y 271.821,Z 875.396,A -85,B 0,C 180,E1 12723.481,E2 12723.481} C_VEL
LIN {X 0,Y 269.648,Z 880.259,A -85,B 0,C 180,E1 12720.234,E2 12720.234} C_VEL
LIN {X 0,Y 268.06,Z 883.367,A -85,B 0,C 180,E1 12716.823,E2 12716.823} C_VEL
LIN {X 0,Y 267.092,Z 884.737,A -85,B 0,C 180,E1 12713.374,E2 12713.374} C_VEL
LIN {X 0,Y 266.666,Z 884.364,A -85,B 0,C 180,E1 12709.946,E2 12709.946} C_VEL
LIN {X 0,Y 266.747,Z 882.143,A -85,B 0,C 180,E1 12706.323,E2 12706.323} C_VEL
LIN {X 0,Y 267.317,Z 878.258,A -85,B 0,C 180,E1 12702.965,E2 12702.965} C_VEL
LIN {X 0,Y 268.408,Z 872.549,A -85,B 0,C 180,E1 12699.647,E2 12699.647} C_VEL
LIN {X 0,Y 269.945,Z 865.31,A -85,B 0,C 180,E1 12696.59,E2 12696.59} C_VEL
LIN {X 0,Y 272.028,Z 855.948,A -85,B 0,C 180,E1 12693.58,E2 12693.58} C_VEL
LIN {X 0,Y 274.224,Z 845.739,A -85,B 0,C 180,E1 12691.042,E2 12691.042} C_VEL
LIN {X 0,Y 276.688,Z 833.592,A -85,B 0,C 180,E1 12688.652,E2 12688.652} C_VEL
LIN {X 0,Y 279.096,Z 820.207,A -85,B 0,C 180,E1 12686.609,E2 12686.609} C_VEL
LIN {X 0,Y 281.207,Z 806.748,A -85,B 0,C 180,E1 12685,E2 12685} C_VEL
LIN {X 0,Y 283.138,Z 791.105,A -85,B 0,C 180,E1 12683.595,E2 12683.595} C_VEL
LIN {X 0,Y 284.558,Z 775.226,A -85,B 0,C 180,E1 12682.573,E2 12682.573} C_VEL
LIN {X 0,Y 285.473,Z 757.62,A -85,B 0,C 180,E1 12681.862,E2 12681.862} C_VEL
LIN {X 0,Y 288.626,Z 673.002,A -85,B 0,C 180,E1 12679.687,E2 12679.687} C_VEL
LIN {X 0,Y 282.056,Z 627.904,A -85,B 0,C 180,E1 12677.51,E2 12677.51} C_VEL
LIN {X 0,Y 285.831,Z 608.302,A -85,B 0,C 180,E1 12673.644,E2 12673.644} C_VEL
LIN {X 0,Y 282.435,Z 593.69,A -85,B 0,C 180,E1 12669.743,E2 12669.743} C_VEL
LIN {X 0,Y 278.573,Z 579.66,A -85,B 0,C 180,E1 12665.621,E2 12665.621} C_VEL
LIN {X 0,Y 274.733,Z 567.674,A -85,B 0,C 180,E1 12661.732,E2 12661.732} C_VEL
LIN {X 0,Y 270.795,Z 556.577,A -85,B 0,C 180,E1 12657.731,E2 12657.731} C_VEL
LIN {X 0,Y 267.269,Z 548.198,A -85,B 0,C 180,E1 12654.296,E2 12654.296} C_VEL
LIN {X 0,Y 266.496,Z 545.687,A -85,B 0,C 180,E1 12653.195,E2 12653.195} C_VEL
LIN {X 0,Y 266.492,Z 545.573,A -85,B 0,C 180,E1 12648.388,E2 12648.388} C_VEL
LIN {X 0,Y 266.476,Z 545.594,A -85,B 0,C 180,E1 12643.602,E2 12643.602} C_VEL
LIN {X 0,Y 266.495,Z 545.589,A -85,B 0,C 180,E1 12638.705,E2 12638.705} C_VEL
LIN {X 0,Y 266.48,Z 545.568,A -85,B 0,C 180,E1 12635.561,E2 12635.561} C_VEL
LIN {X 0,Y 265.469,Z 545.686,A -85,B 0,C 180,E1 12633.905,E2 12633.905} C_VEL
LIN {X 0,Y 261.25,Z 546.248,A -85,B 0,C 180,E1 12630.998,E2 12630.998} C_VEL
LIN {X 0,Y 258.77,Z 546.543,A -85,B 0,C 180,E1 12628.706,E2 12628.706} C_VEL
LIN {X 0,Y 258.569,Z 546.551,A -85,B 0,C 180,E1 12627.961,E2 12627.961} C_VEL
LIN {X 0,Y 258.547,Z 546.58,A -85,B 0,C 180,E1 12622.992,E2 12622.992} C_VEL
LIN {X 0,Y 258.563,Z 546.531,A -85,B 0,C 180,E1 12617.965,E2 12617.965} C_VEL
LIN {X 0,Y 258.567,Z 546.589,A -85,B 0,C 180,E1 12613.189,E2 12613.189} C_VEL
LIN {X 0,Y 258.55,Z 546.531,A -85,B 0,C 180,E1 12608.127,E2 12608.127} C_VEL
LIN {X 0,Y 258.574,Z 546.572,A -85,B 0,C 180,E1 12603.326,E2 12603.326} C_VEL
LIN {X 0,Y 258.557,Z 546.55,A -85,B 0,C 180,E1 12598.449,E2 12598.449} C_VEL
LIN {X 0,Y 258.561,Z 546.547,A -85,B 0,C 180,E1 12593.562,E2 12593.562} C_VEL
LIN {X 0,Y 258.581,Z 546.589,A -85,B 0,C 180,E1 12588.627,E2 12588.627} C_VEL
LIN {X 0,Y 258.562,Z 546.557,A -85,B 0,C 180,E1 12583.834,E2 12583.834} C_VEL
LIN {X 0,Y 258.577,Z 546.552,A -85,B 0,C 180,E1 12578.924,E2 12578.924} C_VEL
LIN {X 0,Y 258.63,Z 546.861,A -85,B 0,C 180,E1 12574.465,E2 12574.465} C_VEL
LIN {X 0,Y 260.314,Z 550.67,A -85,B 0,C 180,E1 12572.802,E2 12572.802} C_VEL
LIN {X 0,Y 264.485,Z 560.453,A -85,B 0,C 180,E1 12569.061,E2 12569.061} C_VEL
LIN {X 0,Y 269.205,Z 571.919,A -85,B 0,C 180,E1 12565.164,E2 12565.164} C_VEL
LIN {X 0,Y 273.984,Z 584.878,A -85,B 0,C 180,E1 12561.346,E2 12561.346} C_VEL
LIN {X 0,Y 278.895,Z 599.684,A -85,B 0,C 180,E1 12557.485,E2 12557.485} C_VEL
LIN {X 0,Y 283.977,Z 616.91,A -85,B 0,C 180,E1 12553.506,E2 12553.506} C_VEL
LIN {X 0,Y 284.3,Z 619.064,A -85,B 0,C 180,E1 12553.09,E2 12553.09} C_VEL
LIN {X 0,Y 285.168,Z 633.59,A -85,B 0,C 180,E1 12552.481,E2 12552.481} C_VEL
LIN {X 0,Y 286.858,Z 657.587,A -85,B 0,C 180,E1 12551.567,E2 12551.567} C_VEL
LIN {X 0,Y 281.194,Z 804.199,A -85,B 0,C 180,E1 12548.026,E2 12548.026} C_VEL
LIN {X 0,Y 279.613,Z 822.478,A -85,B 0,C 180,E1 12547.244,E2 12547.244} C_VEL
LIN {X 0,Y 277.263,Z 840.32,A -85,B 0,C 180,E1 12546.121,E2 12546.121} C_VEL
LIN {X 0,Y 274.436,Z 857.524,A -85,B 0,C 180,E1 12544.635,E2 12544.635} C_VEL
LIN {X 0,Y 271.366,Z 873.805,A -85,B 0,C 180,E1 12542.794,E2 12542.794} C_VEL
LIN {X 0,Y 268.186,Z 889.064,A -85,B 0,C 180,E1 12540.591,E2 12540.591} C_VEL
LIN {X 0,Y 265.066,Z 903.249,A -85,B 0,C 180,E1 12538.034,E2 12538.034} C_VEL
LIN {X 0,Y 262.213,Z 916.602,A -85,B 0,C 180,E1 12535.041,E2 12535.041} C_VEL
LIN {X 0,Y 259.961,Z 927.901,A -85,B 0,C 180,E1 12531.907,E2 12531.907} C_VEL
LIN {X 0,Y 258.325,Z 937.807,A -85,B 0,C 180,E1 12528.506,E2 12528.506} C_VEL
LIN {X 0,Y 257.407,Z 946.276,A -85,B 0,C 180,E1 12524.856,E2 12524.856} C_VEL
LIN {X 0,Y 257.219,Z 953.163,A -85,B 0,C 180,E1 12520.982,E2 12520.982} C_VEL
LIN {X 0,Y 257.592,Z 957.898,A -85,B 0,C 180,E1 12517.361,E2 12517.361} C_VEL
LIN {X 0,Y 258.18,Z 961.001,A -85,B 0,C 180,E1 12513.777,E2 12513.777} C_VEL
LIN {X 0,Y 258.476,Z 962.405,A -85,B 0,C 180,E1 12510.446,E2 12510.446} C_VEL
LIN {X 0,Y 258.215,Z 962.42,A -85,B 0,C 180,E1 12507.34,E2 12507.34} C_VEL
LIN {X 0,Y 257.526,Z 960.955,A -85,B 0,C 180,E1 12503.684,E2 12503.684} C_VEL
LIN {X 0,Y 256.98,Z 957.635,A -85,B 0,C 180,E1 12499.694,E2 12499.694} C_VEL
LIN {X 0,Y 257.102,Z 952.331,A -85,B 0,C 180,E1 12495.546,E2 12495.546} C_VEL
LIN {X 0,Y 258.206,Z 945.236,A -85,B 0,C 180,E1 12491.491,E2 12491.491} C_VEL
LIN {X 0,Y 260.317,Z 936.507,A -85,B 0,C 180,E1 12487.656,E2 12487.656} C_VEL
LIN {X 0,Y 263.324,Z 926.226,A -85,B 0,C 180,E1 12484.114,E2 12484.114} C_VEL
LIN {X 0,Y 267.03,Z 914.446,A -85,B 0,C 180,E1 12480.877,E2 12480.877} C_VEL
LIN {X 0,Y 271.374,Z 900.989,A -85,B 0,C 180,E1 12477.932,E2 12477.932} C_VEL
LIN {X 0,Y 275.832,Z 886.727,A -85,B 0,C 180,E1 12475.445,E2 12475.445} C_VEL
LIN {X 0,Y 280.281,Z 871.314,A -85,B 0,C 180,E1 12473.314,E2 12473.314} C_VEL
LIN {X 0,Y 284.264,Z 855.791,A -85,B 0,C 180,E1 12471.644,E2 12471.644} C_VEL
LIN {X 0,Y 287.894,Z 839.255,A -85,B 0,C 180,E1 12470.288,E2 12470.288} C_VEL
LIN {X 0,Y 290.979,Z 821.635,A -85,B 0,C 180,E1 12469.235,E2 12469.235} C_VEL
LIN {X 0,Y 293.155,Z 803.104,A -85,B 0,C 180,E1 12468.474,E2 12468.474} C_VEL
LIN {X 0,Y 295.047,Z 767.806,A -85,B 0,C 180,E1 12467.599,E2 12467.599} C_VEL
LIN {X 0,Y 300.608,Z 656.968,A -85,B 0,C 180,E1 12464.938,E2 12464.938} C_VEL
LIN {X 0,Y 298.78,Z 633.282,A -85,B 0,C 180,E1 12463.736,E2 12463.736} C_VEL
LIN {X 0,Y 291.738,Z 620.657,A -85,B 0,C 180,E1 12461.666,E2 12461.666} C_VEL
LIN {X 0,Y 288.226,Z 609.858,A -85,B 0,C 180,E1 12458.132,E2 12458.132} C_VEL
LIN {X 0,Y 284.596,Z 599.867,A -85,B 0,C 180,E1 12454.202,E2 12454.202} C_VEL
LIN {X 0,Y 281.285,Z 591.841,A -85,B 0,C 180,E1 12450.315,E2 12450.315} C_VEL
LIN {X 0,Y 279.297,Z 587.379,A -85,B 0,C 180,E1 12447.735,E2 12447.735} C_VEL
LIN {X 0,Y 277.975,Z 584.403,A -85,B 0,C 180,E1 12445.8,E2 12445.8} C_VEL
LIN {X 0,Y 276.336,Z 580.644,A -85,B 0,C 180,E1 12443.002,E2 12443.002} C_VEL
LIN {X 0,Y 274.462,Z 576.549,A -85,B 0,C 180,E1 12439.139,E2 12439.139} C_VEL
LIN {X 0,Y 272.443,Z 572.307,A -85,B 0,C 180,E1 12432.505,E2 12432.505} C_VEL
LIN {X 0,Y 271.69,Z 571.444,A -85,B 0,C 180,E1 12427.188,E2 12427.188} C_VEL
LIN {X 0,Y 272.143,Z 572.1,A -85,B 0,C 180,E1 12422.105,E2 12422.105} C_VEL
LIN {X 0,Y 273.84,Z 576.42,A -85,B 0,C 180,E1 12414.972,E2 12414.972} C_VEL
LIN {X 0,Y 275.446,Z 580.634,A -85,B 0,C 180,E1 12410.809,E2 12410.809} C_VEL
LIN {X 0,Y 276.971,Z 584.638,A -85,B 0,C 180,E1 12407.702,E2 12407.702} C_VEL
LIN {X 0,Y 279.134,Z 590.27,A -85,B 0,C 180,E1 12403.989,E2 12403.989} C_VEL
LIN {X 0,Y 281.657,Z 598.088,A -85,B 0,C 180,E1 12399.858,E2 12399.858} C_VEL
LIN {X 0,Y 284.127,Z 606.354,A -85,B 0,C 180,E1 12396.128,E2 12396.128} C_VEL
LIN {X 0,Y 286.547,Z 616.14,A -85,B 0,C 180,E1 12392.349,E2 12392.349} C_VEL
LIN {X 0,Y 288.585,Z 626.882,A -85,B 0,C 180,E1 12388.774,E2 12388.774} C_VEL
LIN {X 0,Y 288.945,Z 630.52,A -85,B 0,C 180,E1 12388.396,E2 12388.396} C_VEL
LIN {X 0,Y 294.187,Z 660.226,A -85,B 0,C 180,E1 12386.095,E2 12386.095} C_VEL
LIN {X 0,Y 297.071,Z 680.872,A -85,B 0,C 180,E1 12384.746,E2 12384.746} C_VEL
LIN {X 0,Y 292.206,Z 766.375,A -85,B 0,C 180,E1 12382.517,E2 12382.517} C_VEL
LIN {X 0,Y 290.716,Z 782.519,A -85,B 0,C 180,E1 12381.759,E2 12381.759} C_VEL
LIN {X 0,Y 288.533,Z 797.989,A -85,B 0,C 180,E1 12380.691,E2 12380.691} C_VEL
LIN {X 0,Y 285.834,Z 812.039,A -85,B 0,C 180,E1 12379.373,E2 12379.373} C_VEL
LIN {X 0,Y 282.339,Z 826.568,A -85,B 0,C 180,E1 12377.584,E2 12377.584} C_VEL
LIN {X 0,Y 278.781,Z 838.865,A -85,B 0,C 180,E1 12375.622,E2 12375.622} C_VEL
LIN {X 0,Y 274.806,Z 850.887,A -85,B 0,C 180,E1 12373.151,E2 12373.151} C_VEL
LIN {X 0,Y 271.059,Z 860.903,A -85,B 0,C 180,E1 12370.475,E2 12370.475} C_VEL
LIN {X 0,Y 267.582,Z 869.382,A -85,B 0,C 180,E1 12367.515,E2 12367.515} C_VEL
LIN {X 0,Y 264.711,Z 875.826,A -85,B 0,C 180,E1 12364.505,E2 12364.505} C_VEL
LIN {X 0,Y 262.16,Z 881.124,A -85,B 0,C 180,E1 12360.983,E2 12360.983} C_VEL
LIN {X 0,Y 260.413,Z 884.378,A -85,B 0,C 180,E1 12357.509,E2 12357.509} C_VEL
LIN {X 0,Y 259.233,Z 885.935,A -85,B 0,C 180,E1 12353.643,E2 12353.643} C_VEL
